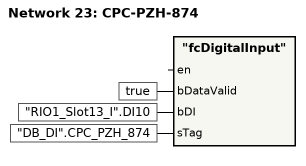
   "fcDigitalInput"(bDataValid := true, bDI := "RIO1_Slot13_I".DI10, sTag := "DB_DI".CPC_PZH_874);
END_REGION
END_FUNCTION_BLOCK

FUNCTION "fcDigitalInput" : Void
{ S7_Optimized_Access := 'TRUE' }
AUTHOR : Heaten
VERSION : 0.1
   VAR_INPUT 
      bDataValid : Bool;   // 1 = valid signal, 0 = invalid signal
      bDI : Bool;   // DI channel
   END_VAR

   VAR_IN_OUT 
      sTag : "stDigitalInput";
   END_VAR


BEGIN
	// Validate a digital input signal
	
	#sTag.bError := NOT(#bDataValid);
	
	IF #sTag.bError = TRUE THEN
	    #sTag.bValue := #sTag.bValueOnError;
	ELSE
	    #sTag.bValue := #bDI;
	END_IF;
END_FUNCTION

FUNCTION "fcAnalogInput" : Void
{ S7_Optimized_Access := 'TRUE' }
AUTHOR : Heaten
VERSION : 0.1
   VAR_INPUT 
      bValidData : Bool;
      iAI : Int;
      fOffset : Real;
   END_VAR

   VAR_OUTPUT 
      fEngValue : Real;
   END_VAR

   VAR_IN_OUT 
      sTag : "stAnalogInput";
   END_VAR

   VAR_TEMP 
      fSlope : Real;
      fIntercept : Real;
      fValue : Real;
   END_VAR


BEGIN
	// This is a version of fbAnalogInput that does not cache the scaling factors
	// An FB version takes 315 bytes per instance :(
	
	#sTag.Raw.iValue := #iAI;
	#sTag.Raw.bFault := NOT #bValidData;
	
	// Scaling
	IF NOT #bValidData THEN
	    #sTag.Eng.bError := TRUE;
	    #sTag.Eng.fValue := "NaN"();
	ELSE
	    #sTag.Eng.bError := FALSE;
	    IF #sTag.Raw.iMax <> 0 OR #sTag.Raw.iMin <> 0 THEN
	        #fSlope := (#sTag.Eng.fMax - #sTag.Eng.fMin) / INT_TO_REAL(#sTag.Raw.iMax - #sTag.Raw.iMin);
	    END_IF;
	    #fIntercept := #sTag.Eng.fMax - #fSlope*INT_TO_REAL(#sTag.Raw.iMax);
	    #fValue := INT_TO_REAL(#iAI)*#fSlope + #fIntercept + #fOffset;
	    // Apply limiting, if enabled
	    "fcCalcAssign"(fValue := #fValue, sTag := #sTag.Eng);
	END_IF;
	
	// Local output
	#fEngValue := #sTag.Eng.fValue;
	
END_FUNCTION

FUNCTION "fcCalcAssign" : Void

{ S7_Optimized_Access := 'TRUE' }
VERSION : 0.1
VAR_INPUT
  fValue : Real;
END_VAR

VAR_OUTPUT

END_VAR

VAR_IN_OUT
  sTag : "stCalcValue";
END_VAR

VAR_TEMP

END_VAR

VAR CONSTANT

END_VAR


BEGIN
	// When assigning to a calc value, set sTag.fValue and bits
	
	IF "isNaN"(#fValue) THEN
	    // Set error on NaN in
	    #sTag.bError := TRUE;
	    #sTag.fValue := #fValue;
	    #sTag.bLimited := FALSE;
	ELSE
	    // Valid values
	    #sTag.bError := FALSE;
	    IF #sTag.bCheckLimits = TRUE THEN
	        // With limitation
	        #sTag.fValue := LIMIT(IN := #fValue, MN := #sTag.fMin, MX := #sTag.fMax);
	        #sTag.bLimited := #fValue <> #sTag.fValue;
	    ELSE
	        // Without limitation
	        #sTag.fValue := #fValue;
	        #sTag.bLimited := FALSE;
	    END_IF;
	END_IF;
END_FUNCTION

FUNCTION "isNaN" : Bool   // FC19, FBD
TITLE = isNaN
{ S7_Optimized_Access := 'TRUE' }
VERSION : 0.1
// Returns TRUE if a REAL is NaN
// stored: AutoNumber true, IsIECCheckEnabled false, SetENOAutomatically false, UDAEnableTagReadback false
   VAR_INPUT
      In : Real;
   END_VAR
BEGIN

REGION Network 1
   // NOT_OK is a compiler builtin, but not available in SCL
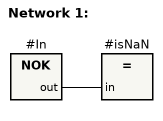
   // no SCL statement known for NOK: written as a call
   #isNaN := NOK(#In);
END_REGION
END_FUNCTION

FUNCTION_BLOCK "AnalogInputProcessing"   // FB37, FBD
TITLE = Handle analog inputs
{ S7_Optimized_Access := 'TRUE' }
AUTHOR : Heaten
VERSION : 0.1
// Map & scale analog inputs
// stored: AutoNumber true, IsIECCheckEnabled false, IsRetainMemResEnabled false, MemoryReserve 0, SetENOAutomatically false, UDAEnableTagReadback false
   VAR
      bHere : Bool;
   END_VAR
   VAR_TEMP
      fDummy : Real;
      fMaxWindingTemperature : Real;
      HBL_PT_05 : Real;
   END_VAR
   VAR_TEMP   // added for the SCL form of the ladder/FBD networks
      _w1 : Bool;
   END_VAR
BEGIN

REGION Network 1: HBL_TT_03 Oil sump oil temperature
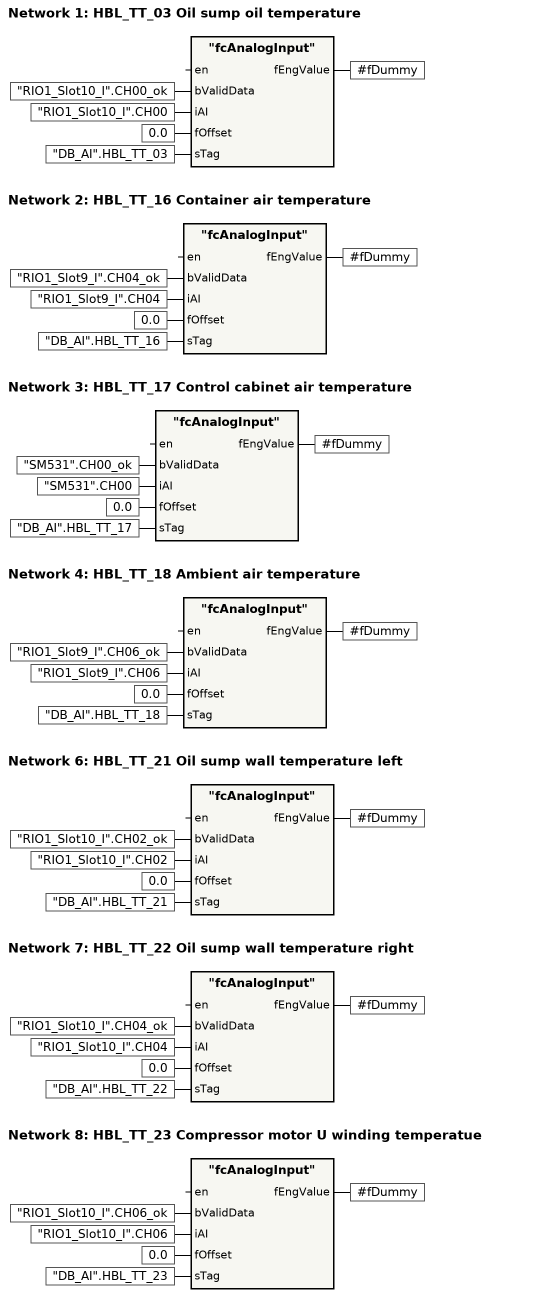
   "fcAnalogInput"(bValidData := "RIO1_Slot10_I".CH00_ok,
                   iAI := "RIO1_Slot10_I".CH00,
                   fOffset := 0.0,
                   sTag := "DB_AI".HBL_TT_03,
                   fEngValue => #fDummy);
END_REGION

REGION Network 2: HBL_TT_16 Container air temperature
   "fcAnalogInput"(bValidData := "RIO1_Slot9_I".CH04_ok,
                   iAI := "RIO1_Slot9_I".CH04,
                   fOffset := 0.0,
                   sTag := "DB_AI".HBL_TT_16,
                   fEngValue => #fDummy);
END_REGION

REGION Network 3: HBL_TT_17 Control cabinet air temperature
   "fcAnalogInput"(bValidData := "SM531".CH00_ok,
                   iAI := "SM531".CH00,
                   fOffset := 0.0,
                   sTag := "DB_AI".HBL_TT_17,
                   fEngValue => #fDummy);
END_REGION

REGION Network 4: HBL_TT_18 Ambient air temperature
   "fcAnalogInput"(bValidData := "RIO1_Slot9_I".CH06_ok,
                   iAI := "RIO1_Slot9_I".CH06,
                   fOffset := 0.0,
                   sTag := "DB_AI".HBL_TT_18,
                   fEngValue => #fDummy);
END_REGION

REGION Network 5: HBL_TT_19 Main inverter temperature
   // ##This is a fieldbus value. get from inverter, if we need it.
END_REGION

REGION Network 6: HBL_TT_21 Oil sump wall temperature left
   "fcAnalogInput"(bValidData := "RIO1_Slot10_I".CH02_ok,
                   iAI := "RIO1_Slot10_I".CH02,
                   fOffset := 0.0,
                   sTag := "DB_AI".HBL_TT_21,
                   fEngValue => #fDummy);
END_REGION

REGION Network 7: HBL_TT_22 Oil sump wall temperature right
   "fcAnalogInput"(bValidData := "RIO1_Slot10_I".CH04_ok,
                   iAI := "RIO1_Slot10_I".CH04,
                   fOffset := 0.0,
                   sTag := "DB_AI".HBL_TT_22,
                   fEngValue => #fDummy);
END_REGION

REGION Network 8: HBL_TT_23 Compressor motor U winding temperatue
   "fcAnalogInput"(bValidData := "RIO1_Slot10_I".CH06_ok,
                   iAI := "RIO1_Slot10_I".CH06,
                   fOffset := 0.0,
                   sTag := "DB_AI".HBL_TT_23,
                   fEngValue => #fDummy);
END_REGION

REGION Network 9: HBL_TT_24 Compressor motor V winding temperature
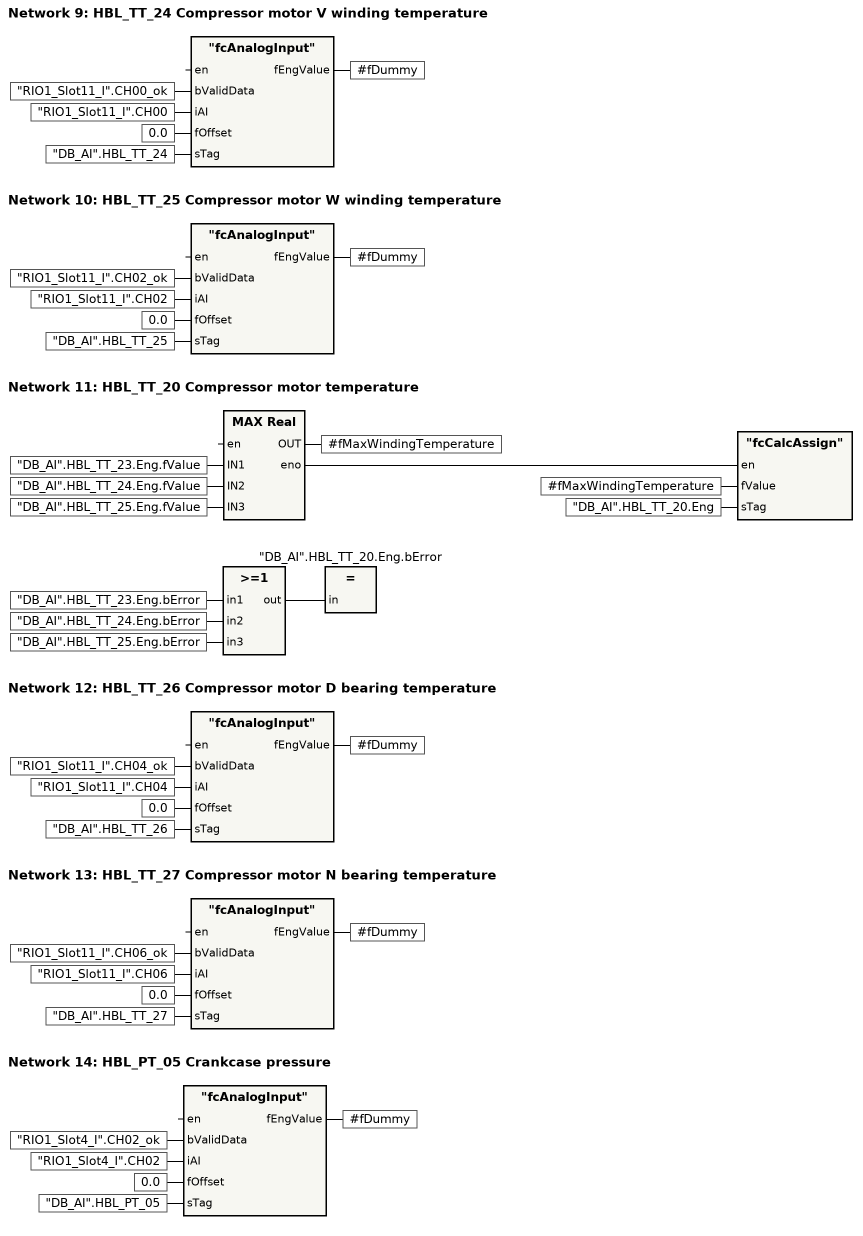
   "fcAnalogInput"(bValidData := "RIO1_Slot11_I".CH00_ok,
                   iAI := "RIO1_Slot11_I".CH00,
                   fOffset := 0.0,
                   sTag := "DB_AI".HBL_TT_24,
                   fEngValue => #fDummy);
END_REGION

REGION Network 10: HBL_TT_25 Compressor motor W winding temperature
   "fcAnalogInput"(bValidData := "RIO1_Slot11_I".CH02_ok,
                   iAI := "RIO1_Slot11_I".CH02,
                   fOffset := 0.0,
                   sTag := "DB_AI".HBL_TT_25,
                   fEngValue => #fDummy);
END_REGION

REGION Network 11: HBL_TT_20 Compressor motor temperature
   // MAX of any of the winding temperatures. If there is only one motor temperature, eg one PTC, use HBL-TT-20 as the analog input object
   // The individual winding temperatures are not used in the program (but are available for monitoring & logging)
   #fMaxWindingTemperature := MAX(IN1 := "DB_AI".HBL_TT_23.Eng.fValue, IN2 := "DB_AI".HBL_TT_24.Eng.fValue, IN3 := "DB_AI".HBL_TT_25.Eng.fValue);
   "fcCalcAssign"(fValue := #fMaxWindingTemperature, sTag := "DB_AI".HBL_TT_20.Eng);
   "DB_AI".HBL_TT_20.Eng.bError := "DB_AI".HBL_TT_23.Eng.bError OR "DB_AI".HBL_TT_24.Eng.bError OR "DB_AI".HBL_TT_25.Eng.bError;
END_REGION

REGION Network 12: HBL_TT_26 Compressor motor D bearing temperature
   "fcAnalogInput"(bValidData := "RIO1_Slot11_I".CH04_ok,
                   iAI := "RIO1_Slot11_I".CH04,
                   fOffset := 0.0,
                   sTag := "DB_AI".HBL_TT_26,
                   fEngValue => #fDummy);
END_REGION

REGION Network 13: HBL_TT_27 Compressor motor N bearing temperature
   "fcAnalogInput"(bValidData := "RIO1_Slot11_I".CH06_ok,
                   iAI := "RIO1_Slot11_I".CH06,
                   fOffset := 0.0,
                   sTag := "DB_AI".HBL_TT_27,
                   fEngValue => #fDummy);
END_REGION

REGION Network 14: HBL_PT_05 Crankcase pressure
   "fcAnalogInput"(bValidData := "RIO1_Slot4_I".CH02_ok,
                   iAI := "RIO1_Slot4_I".CH02,
                   fOffset := 0.0,
                   sTag := "DB_AI".HBL_PT_05,
                   fEngValue => #fDummy);
END_REGION

REGION Network 15: HBL_CT_01 Gas detector
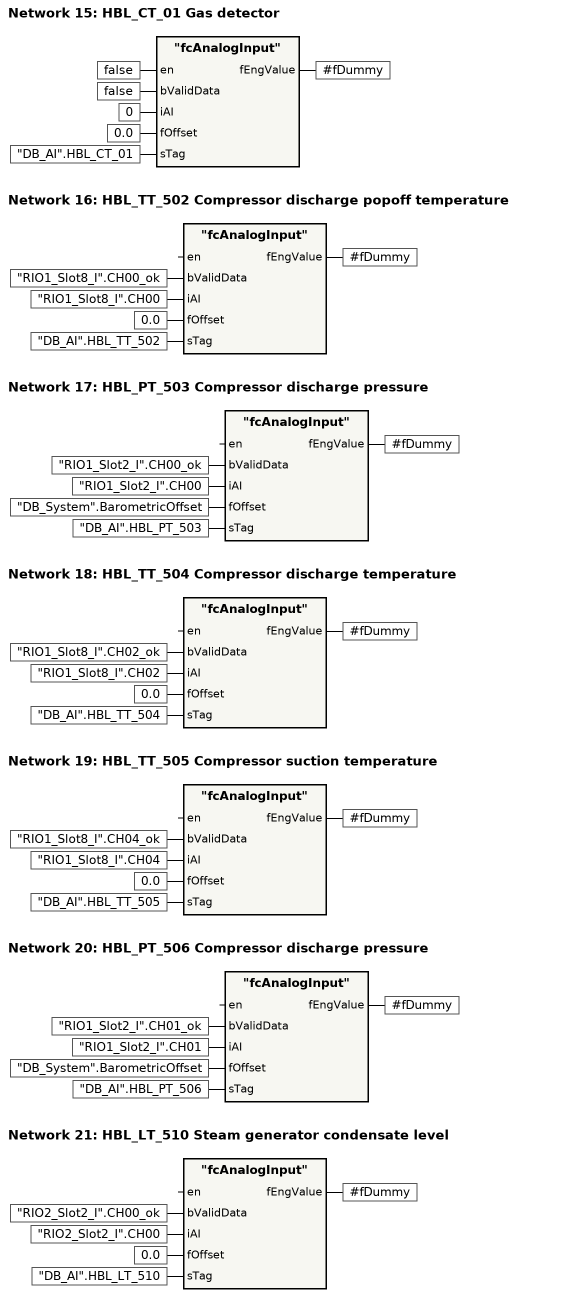
   IF false THEN
       "fcAnalogInput"(bValidData := false,
                       iAI := 0,
                       fOffset := 0.0,
                       sTag := "DB_AI".HBL_CT_01,
                       fEngValue => #fDummy);
   END_IF;
END_REGION

REGION Network 16: HBL_TT_502 Compressor discharge popoff temperature
   "fcAnalogInput"(bValidData := "RIO1_Slot8_I".CH00_ok,
                   iAI := "RIO1_Slot8_I".CH00,
                   fOffset := 0.0,
                   sTag := "DB_AI".HBL_TT_502,
                   fEngValue => #fDummy);
END_REGION

REGION Network 17: HBL_PT_503 Compressor discharge pressure
   "fcAnalogInput"(bValidData := "RIO1_Slot2_I".CH00_ok,
                   iAI := "RIO1_Slot2_I".CH00,
                   fOffset := "DB_System".BarometricOffset,
                   sTag := "DB_AI".HBL_PT_503,
                   fEngValue => #fDummy);
END_REGION

REGION Network 18: HBL_TT_504 Compressor discharge temperature
   "fcAnalogInput"(bValidData := "RIO1_Slot8_I".CH02_ok,
                   iAI := "RIO1_Slot8_I".CH02,
                   fOffset := 0.0,
                   sTag := "DB_AI".HBL_TT_504,
                   fEngValue => #fDummy);
END_REGION

REGION Network 19: HBL_TT_505 Compressor suction temperature
   "fcAnalogInput"(bValidData := "RIO1_Slot8_I".CH04_ok,
                   iAI := "RIO1_Slot8_I".CH04,
                   fOffset := 0.0,
                   sTag := "DB_AI".HBL_TT_505,
                   fEngValue => #fDummy);
END_REGION

REGION Network 20: HBL_PT_506 Compressor discharge pressure
   "fcAnalogInput"(bValidData := "RIO1_Slot2_I".CH01_ok,
                   iAI := "RIO1_Slot2_I".CH01,
                   fOffset := "DB_System".BarometricOffset,
                   sTag := "DB_AI".HBL_PT_506,
                   fEngValue => #fDummy);
END_REGION

REGION Network 21: HBL_LT_510 Steam generator condensate level
   "fcAnalogInput"(bValidData := "RIO2_Slot2_I".CH00_ok,
                   iAI := "RIO2_Slot2_I".CH00,
                   fOffset := 0.0,
                   sTag := "DB_AI".HBL_LT_510,
                   fEngValue => #fDummy);
END_REGION

REGION Network 22: HBL_PT_511 Heat sink discharge pressure
   // Local or remote
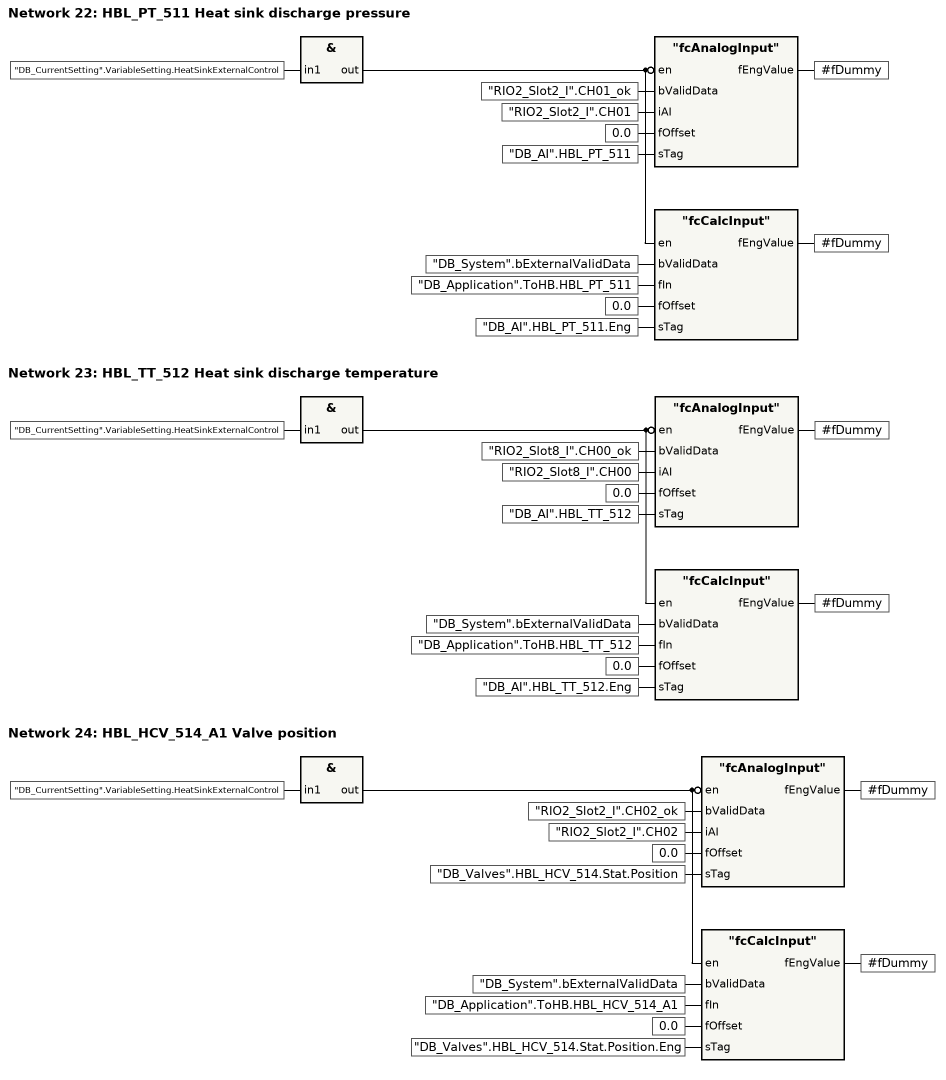
   #_w1 := "DB_CurrentSetting".VariableSetting.HeatSinkExternalControl;
   IF NOT "DB_CurrentSetting".VariableSetting.HeatSinkExternalControl THEN
       "fcAnalogInput"(bValidData := "RIO2_Slot2_I".CH01_ok,
                       iAI := "RIO2_Slot2_I".CH01,
                       fOffset := 0.0,
                       sTag := "DB_AI".HBL_PT_511,
                       fEngValue => #fDummy);
   END_IF;
   IF #_w1 THEN
       "fcCalcInput"(bValidData := "DB_System".bExternalValidData,
                     fIn := "DB_Application".ToHB.HBL_PT_511,
                     fOffset := 0.0,
                     sTag := "DB_AI".HBL_PT_511.Eng,
                     fEngValue => #fDummy);
   END_IF;
END_REGION

REGION Network 23: HBL_TT_512 Heat sink discharge temperature
   // Local or remote
   #_w1 := "DB_CurrentSetting".VariableSetting.HeatSinkExternalControl;
   IF NOT "DB_CurrentSetting".VariableSetting.HeatSinkExternalControl THEN
       "fcAnalogInput"(bValidData := "RIO2_Slot8_I".CH00_ok,
                       iAI := "RIO2_Slot8_I".CH00,
                       fOffset := 0.0,
                       sTag := "DB_AI".HBL_TT_512,
                       fEngValue => #fDummy);
   END_IF;
   IF #_w1 THEN
       "fcCalcInput"(bValidData := "DB_System".bExternalValidData,
                     fIn := "DB_Application".ToHB.HBL_TT_512,
                     fOffset := 0.0,
                     sTag := "DB_AI".HBL_TT_512.Eng,
                     fEngValue => #fDummy);
   END_IF;
END_REGION

REGION Network 24: HBL_HCV_514_A1 Valve position
   // Local or remote
   #_w1 := "DB_CurrentSetting".VariableSetting.HeatSinkExternalControl;
   IF NOT "DB_CurrentSetting".VariableSetting.HeatSinkExternalControl THEN
       "fcAnalogInput"(bValidData := "RIO2_Slot2_I".CH02_ok,
                       iAI := "RIO2_Slot2_I".CH02,
                       fOffset := 0.0,
                       sTag := "DB_Valves".HBL_HCV_514.Stat.Position,
                       fEngValue => #fDummy);
   END_IF;
   IF #_w1 THEN
       "fcCalcInput"(bValidData := "DB_System".bExternalValidData,
                     fIn := "DB_Application".ToHB.HBL_HCV_514_A1,
                     fOffset := 0.0,
                     sTag := "DB_Valves".HBL_HCV_514.Stat.Position.Eng,
                     fEngValue => #fDummy);
   END_IF;
END_REGION

REGION Network 25: HBL_HCV_515_A1 Heat sink condensate blowdown valve position
   // Local or remote
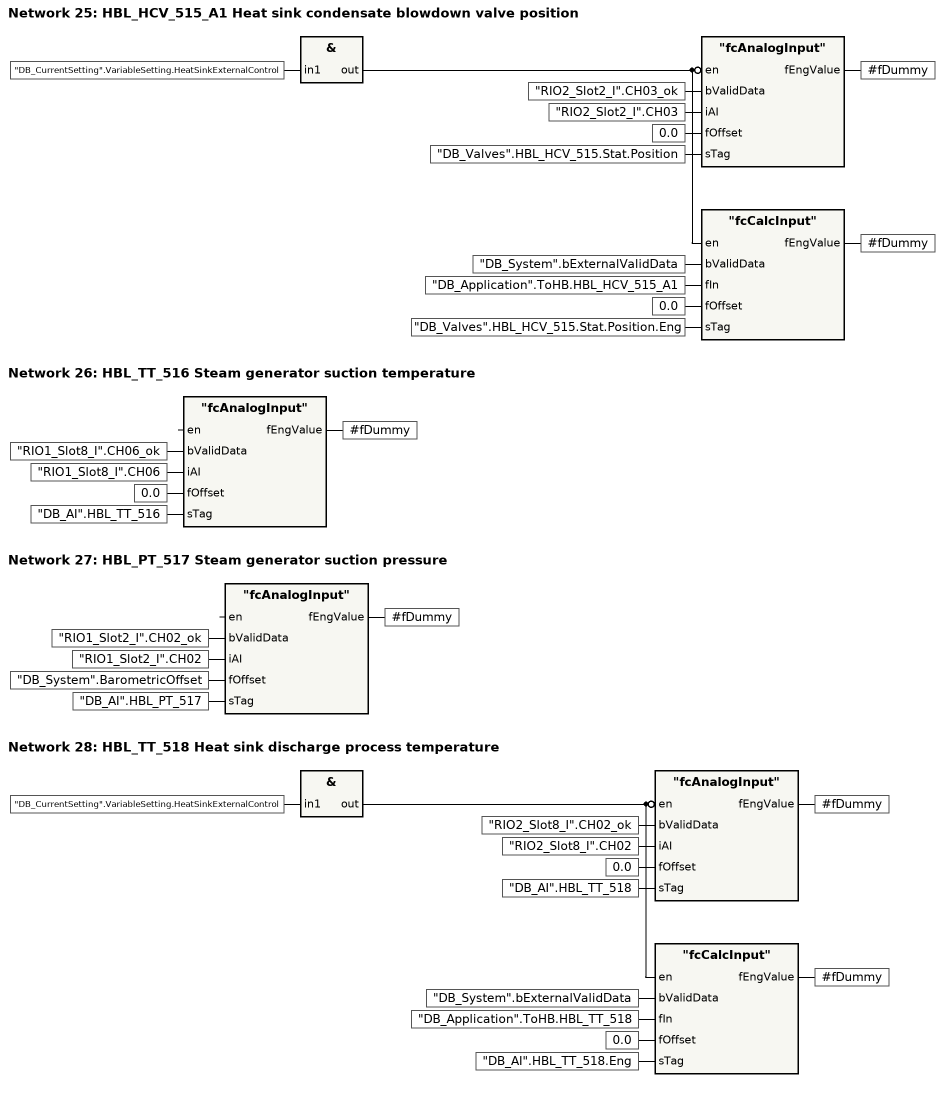
   #_w1 := "DB_CurrentSetting".VariableSetting.HeatSinkExternalControl;
   IF NOT "DB_CurrentSetting".VariableSetting.HeatSinkExternalControl THEN
       "fcAnalogInput"(bValidData := "RIO2_Slot2_I".CH03_ok,
                       iAI := "RIO2_Slot2_I".CH03,
                       fOffset := 0.0,
                       sTag := "DB_Valves".HBL_HCV_515.Stat.Position,
                       fEngValue => #fDummy);
   END_IF;
   IF #_w1 THEN
       "fcCalcInput"(bValidData := "DB_System".bExternalValidData,
                     fIn := "DB_Application".ToHB.HBL_HCV_515_A1,
                     fOffset := 0.0,
                     sTag := "DB_Valves".HBL_HCV_515.Stat.Position.Eng,
                     fEngValue => #fDummy);
   END_IF;
END_REGION

REGION Network 26: HBL_TT_516 Steam generator suction temperature
   "fcAnalogInput"(bValidData := "RIO1_Slot8_I".CH06_ok,
                   iAI := "RIO1_Slot8_I".CH06,
                   fOffset := 0.0,
                   sTag := "DB_AI".HBL_TT_516,
                   fEngValue => #fDummy);
END_REGION

REGION Network 27: HBL_PT_517 Steam generator suction pressure
   "fcAnalogInput"(bValidData := "RIO1_Slot2_I".CH02_ok,
                   iAI := "RIO1_Slot2_I".CH02,
                   fOffset := "DB_System".BarometricOffset,
                   sTag := "DB_AI".HBL_PT_517,
                   fEngValue => #fDummy);
END_REGION

REGION Network 28: HBL_TT_518 Heat sink discharge process temperature
   // Local or remote
   #_w1 := "DB_CurrentSetting".VariableSetting.HeatSinkExternalControl;
   IF NOT "DB_CurrentSetting".VariableSetting.HeatSinkExternalControl THEN
       "fcAnalogInput"(bValidData := "RIO2_Slot8_I".CH02_ok,
                       iAI := "RIO2_Slot8_I".CH02,
                       fOffset := 0.0,
                       sTag := "DB_AI".HBL_TT_518,
                       fEngValue => #fDummy);
   END_IF;
   IF #_w1 THEN
       "fcCalcInput"(bValidData := "DB_System".bExternalValidData,
                     fIn := "DB_Application".ToHB.HBL_TT_518,
                     fOffset := 0.0,
                     sTag := "DB_AI".HBL_TT_518.Eng,
                     fEngValue => #fDummy);
   END_IF;
END_REGION

REGION Network 29: HBL_PT_519 Heat sink discharge process pressure
   // Local or remote
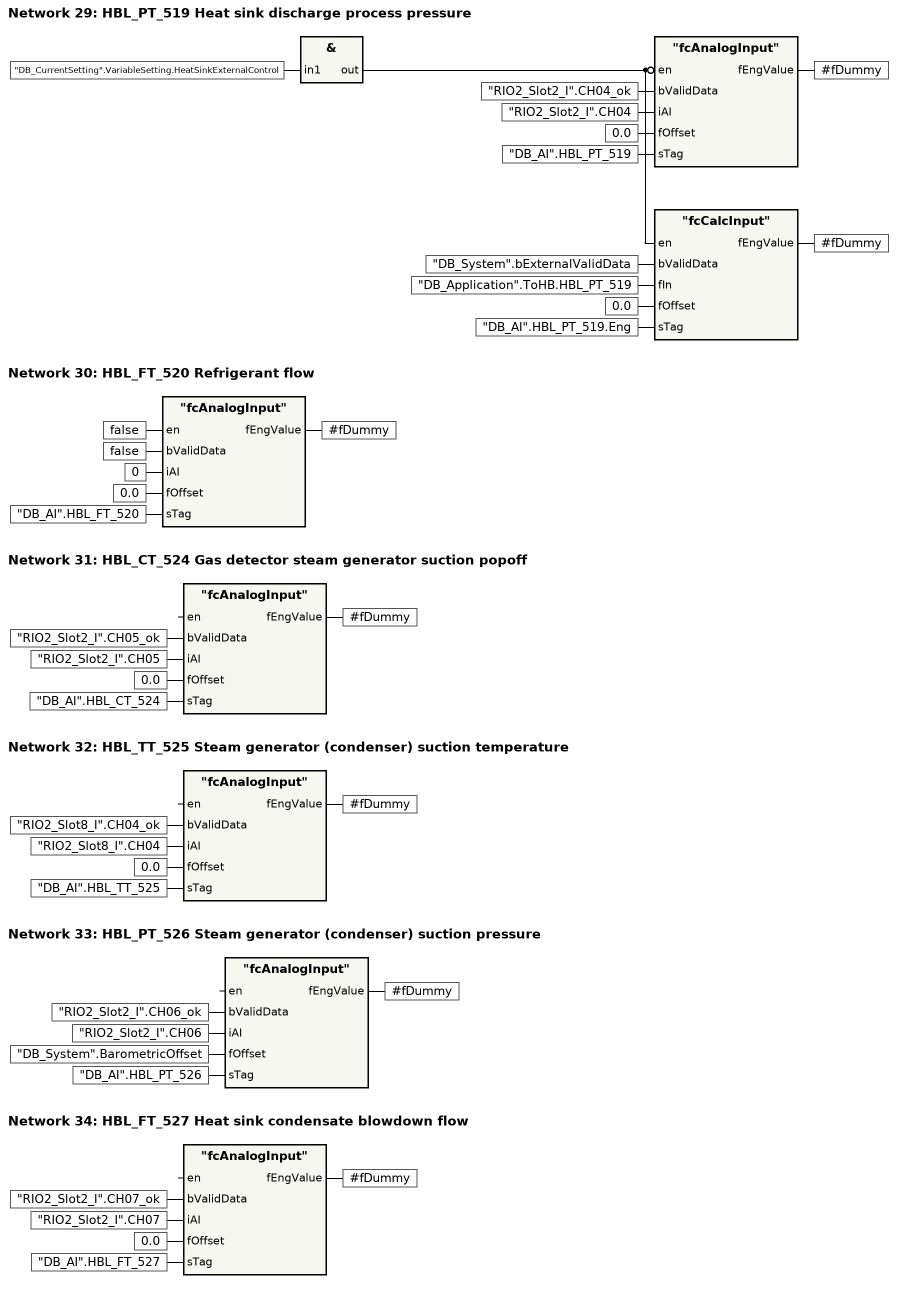
   #_w1 := "DB_CurrentSetting".VariableSetting.HeatSinkExternalControl;
   IF NOT "DB_CurrentSetting".VariableSetting.HeatSinkExternalControl THEN
       "fcAnalogInput"(bValidData := "RIO2_Slot2_I".CH04_ok,
                       iAI := "RIO2_Slot2_I".CH04,
                       fOffset := 0.0,
                       sTag := "DB_AI".HBL_PT_519,
                       fEngValue => #fDummy);
   END_IF;
   IF #_w1 THEN
       "fcCalcInput"(bValidData := "DB_System".bExternalValidData,
                     fIn := "DB_Application".ToHB.HBL_PT_519,
                     fOffset := 0.0,
                     sTag := "DB_AI".HBL_PT_519.Eng,
                     fEngValue => #fDummy);
   END_IF;
END_REGION

REGION Network 30: HBL_FT_520 Refrigerant flow
   // Not used in Offenau
   IF false THEN
       "fcAnalogInput"(bValidData := false,
                       iAI := 0,
                       fOffset := 0.0,
                       sTag := "DB_AI".HBL_FT_520,
                       fEngValue => #fDummy);
   END_IF;
END_REGION

REGION Network 31: HBL_CT_524 Gas detector steam generator suction popoff
   "fcAnalogInput"(bValidData := "RIO2_Slot2_I".CH05_ok,
                   iAI := "RIO2_Slot2_I".CH05,
                   fOffset := 0.0,
                   sTag := "DB_AI".HBL_CT_524,
                   fEngValue => #fDummy);
END_REGION

REGION Network 32: HBL_TT_525 Steam generator (condenser) suction temperature
   "fcAnalogInput"(bValidData := "RIO2_Slot8_I".CH04_ok,
                   iAI := "RIO2_Slot8_I".CH04,
                   fOffset := 0.0,
                   sTag := "DB_AI".HBL_TT_525,
                   fEngValue => #fDummy);
END_REGION

REGION Network 33: HBL_PT_526 Steam generator (condenser) suction pressure
   "fcAnalogInput"(bValidData := "RIO2_Slot2_I".CH06_ok,
                   iAI := "RIO2_Slot2_I".CH06,
                   fOffset := "DB_System".BarometricOffset,
                   sTag := "DB_AI".HBL_PT_526,
                   fEngValue => #fDummy);
END_REGION

REGION Network 34: HBL_FT_527 Heat sink condensate blowdown flow
   "fcAnalogInput"(bValidData := "RIO2_Slot2_I".CH07_ok,
                   iAI := "RIO2_Slot2_I".CH07,
                   fOffset := 0.0,
                   sTag := "DB_AI".HBL_FT_527,
                   fEngValue => #fDummy);
END_REGION

REGION Network 35: HBL_TT_530 Expansion valve B discharge temperature
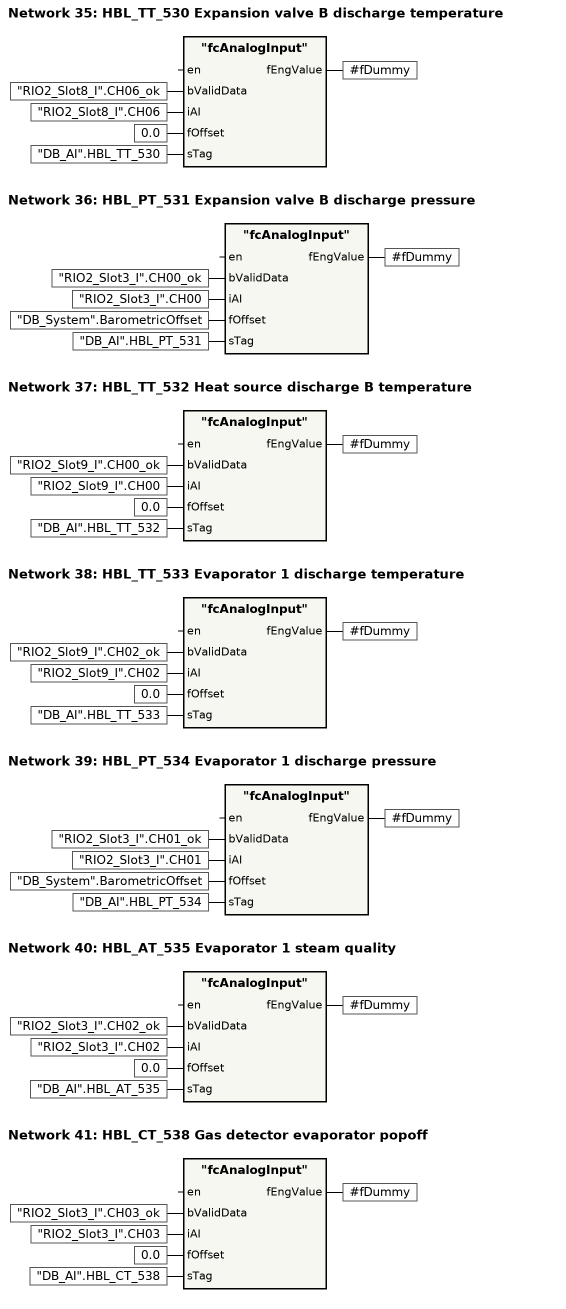
   "fcAnalogInput"(bValidData := "RIO2_Slot8_I".CH06_ok,
                   iAI := "RIO2_Slot8_I".CH06,
                   fOffset := 0.0,
                   sTag := "DB_AI".HBL_TT_530,
                   fEngValue => #fDummy);
END_REGION

REGION Network 36: HBL_PT_531 Expansion valve B discharge pressure
   // Convert from rel to abs
   "fcAnalogInput"(bValidData := "RIO2_Slot3_I".CH00_ok,
                   iAI := "RIO2_Slot3_I".CH00,
                   fOffset := "DB_System".BarometricOffset,
                   sTag := "DB_AI".HBL_PT_531,
                   fEngValue => #fDummy);
END_REGION

REGION Network 37: HBL_TT_532 Heat source discharge B temperature
   "fcAnalogInput"(bValidData := "RIO2_Slot9_I".CH00_ok,
                   iAI := "RIO2_Slot9_I".CH00,
                   fOffset := 0.0,
                   sTag := "DB_AI".HBL_TT_532,
                   fEngValue => #fDummy);
END_REGION

REGION Network 38: HBL_TT_533 Evaporator 1 discharge temperature
   "fcAnalogInput"(bValidData := "RIO2_Slot9_I".CH02_ok,
                   iAI := "RIO2_Slot9_I".CH02,
                   fOffset := 0.0,
                   sTag := "DB_AI".HBL_TT_533,
                   fEngValue => #fDummy);
END_REGION

REGION Network 39: HBL_PT_534 Evaporator 1 discharge pressure
   // Convert from rel to abs
   "fcAnalogInput"(bValidData := "RIO2_Slot3_I".CH01_ok,
                   iAI := "RIO2_Slot3_I".CH01,
                   fOffset := "DB_System".BarometricOffset,
                   sTag := "DB_AI".HBL_PT_534,
                   fEngValue => #fDummy);
END_REGION

REGION Network 40: HBL_AT_535 Evaporator 1 steam quality
   "fcAnalogInput"(bValidData := "RIO2_Slot3_I".CH02_ok,
                   iAI := "RIO2_Slot3_I".CH02,
                   fOffset := 0.0,
                   sTag := "DB_AI".HBL_AT_535,
                   fEngValue => #fDummy);
END_REGION

REGION Network 41: HBL_CT_538 Gas detector evaporator popoff
   "fcAnalogInput"(bValidData := "RIO2_Slot3_I".CH03_ok,
                   iAI := "RIO2_Slot3_I".CH03,
                   fOffset := 0.0,
                   sTag := "DB_AI".HBL_CT_538,
                   fEngValue => #fDummy);
END_REGION

REGION Network 42: HBL_TT_540 Expansion valve A discharge temperature
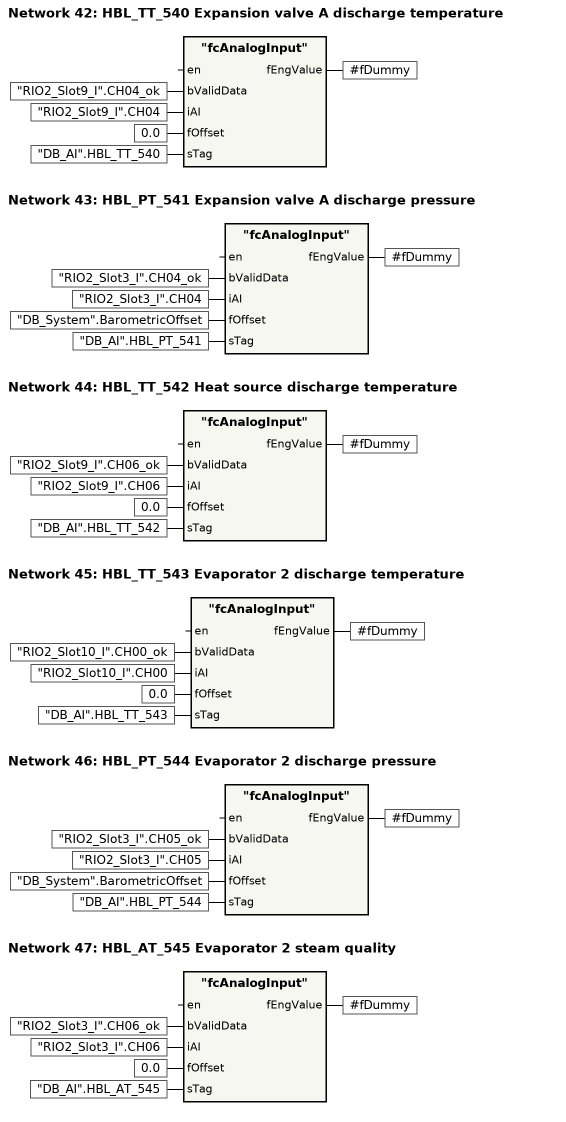
   "fcAnalogInput"(bValidData := "RIO2_Slot9_I".CH04_ok,
                   iAI := "RIO2_Slot9_I".CH04,
                   fOffset := 0.0,
                   sTag := "DB_AI".HBL_TT_540,
                   fEngValue => #fDummy);
END_REGION

REGION Network 43: HBL_PT_541 Expansion valve A discharge pressure
   "fcAnalogInput"(bValidData := "RIO2_Slot3_I".CH04_ok,
                   iAI := "RIO2_Slot3_I".CH04,
                   fOffset := "DB_System".BarometricOffset,
                   sTag := "DB_AI".HBL_PT_541,
                   fEngValue => #fDummy);
END_REGION

REGION Network 44: HBL_TT_542 Heat source discharge temperature
   "fcAnalogInput"(bValidData := "RIO2_Slot9_I".CH06_ok,
                   iAI := "RIO2_Slot9_I".CH06,
                   fOffset := 0.0,
                   sTag := "DB_AI".HBL_TT_542,
                   fEngValue => #fDummy);
END_REGION

REGION Network 45: HBL_TT_543 Evaporator 2 discharge temperature
   "fcAnalogInput"(bValidData := "RIO2_Slot10_I".CH00_ok,
                   iAI := "RIO2_Slot10_I".CH00,
                   fOffset := 0.0,
                   sTag := "DB_AI".HBL_TT_543,
                   fEngValue => #fDummy);
END_REGION

REGION Network 46: HBL_PT_544 Evaporator 2 discharge pressure
   "fcAnalogInput"(bValidData := "RIO2_Slot3_I".CH05_ok,
                   iAI := "RIO2_Slot3_I".CH05,
                   fOffset := "DB_System".BarometricOffset,
                   sTag := "DB_AI".HBL_PT_544,
                   fEngValue => #fDummy);
END_REGION

REGION Network 47: HBL_AT_545 Evaporator 2 steam quality
   "fcAnalogInput"(bValidData := "RIO2_Slot3_I".CH06_ok,
                   iAI := "RIO2_Slot3_I".CH06,
                   fOffset := 0.0,
                   sTag := "DB_AI".HBL_AT_545,
                   fEngValue => #fDummy);
END_REGION

REGION Network 48: HBL_TT_546 Heat source suction temperature
   // Local or remote
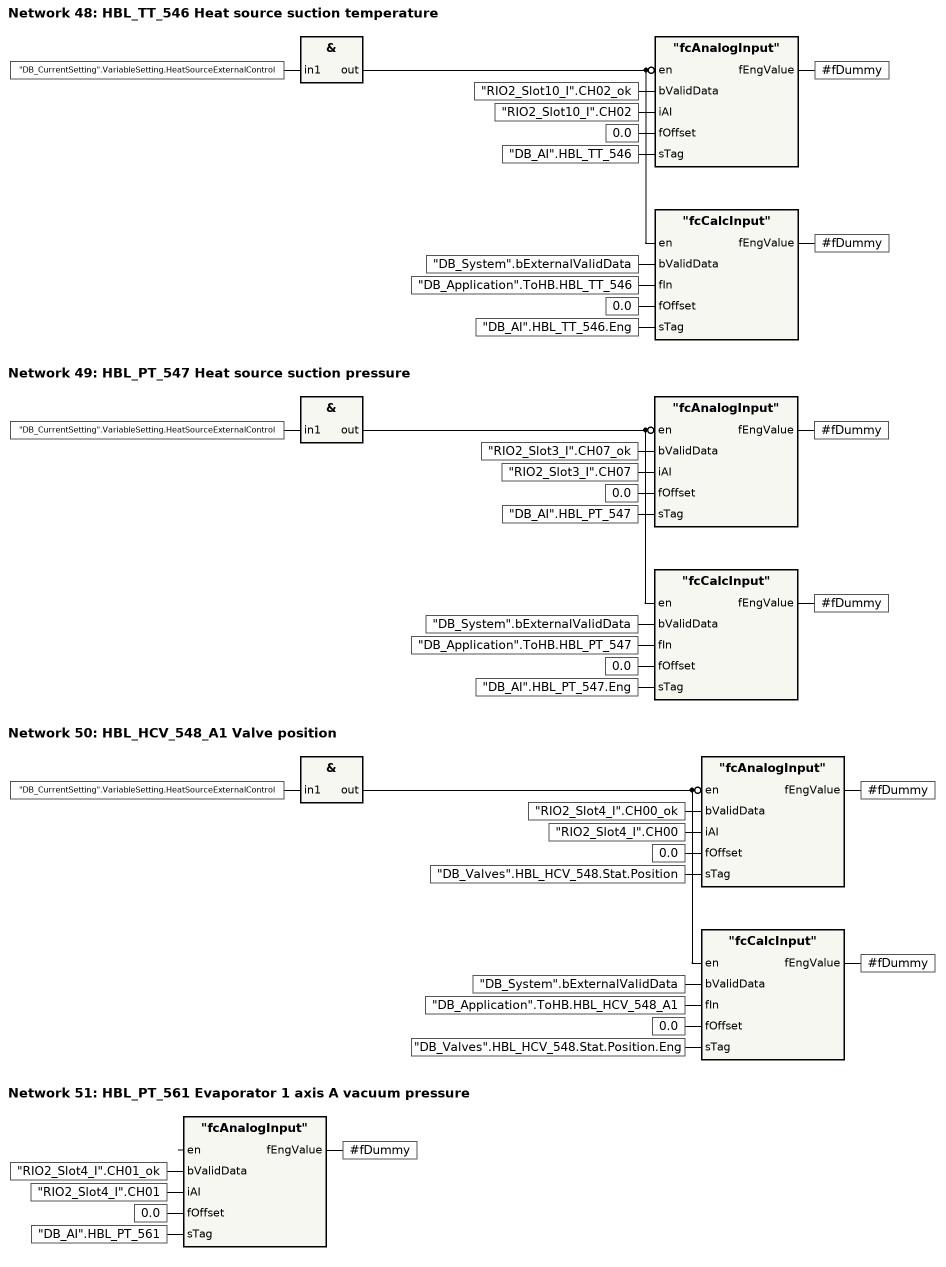
   #_w1 := "DB_CurrentSetting".VariableSetting.HeatSourceExternalControl;
   IF NOT "DB_CurrentSetting".VariableSetting.HeatSourceExternalControl THEN
       "fcAnalogInput"(bValidData := "RIO2_Slot10_I".CH02_ok,
                       iAI := "RIO2_Slot10_I".CH02,
                       fOffset := 0.0,
                       sTag := "DB_AI".HBL_TT_546,
                       fEngValue => #fDummy);
   END_IF;
   IF #_w1 THEN
       "fcCalcInput"(bValidData := "DB_System".bExternalValidData,
                     fIn := "DB_Application".ToHB.HBL_TT_546,
                     fOffset := 0.0,
                     sTag := "DB_AI".HBL_TT_546.Eng,
                     fEngValue => #fDummy);
   END_IF;
END_REGION

REGION Network 49: HBL_PT_547 Heat source suction pressure
   // Local or remote
   #_w1 := "DB_CurrentSetting".VariableSetting.HeatSourceExternalControl;
   IF NOT "DB_CurrentSetting".VariableSetting.HeatSourceExternalControl THEN
       "fcAnalogInput"(bValidData := "RIO2_Slot3_I".CH07_ok,
                       iAI := "RIO2_Slot3_I".CH07,
                       fOffset := 0.0,
                       sTag := "DB_AI".HBL_PT_547,
                       fEngValue => #fDummy);
   END_IF;
   IF #_w1 THEN
       "fcCalcInput"(bValidData := "DB_System".bExternalValidData,
                     fIn := "DB_Application".ToHB.HBL_PT_547,
                     fOffset := 0.0,
                     sTag := "DB_AI".HBL_PT_547.Eng,
                     fEngValue => #fDummy);
   END_IF;
END_REGION

REGION Network 50: HBL_HCV_548_A1 Valve position
   // Local or remote
   #_w1 := "DB_CurrentSetting".VariableSetting.HeatSourceExternalControl;
   IF NOT "DB_CurrentSetting".VariableSetting.HeatSourceExternalControl THEN
       "fcAnalogInput"(bValidData := "RIO2_Slot4_I".CH00_ok,
                       iAI := "RIO2_Slot4_I".CH00,
                       fOffset := 0.0,
                       sTag := "DB_Valves".HBL_HCV_548.Stat.Position,
                       fEngValue => #fDummy);
   END_IF;
   IF #_w1 THEN
       "fcCalcInput"(bValidData := "DB_System".bExternalValidData,
                     fIn := "DB_Application".ToHB.HBL_HCV_548_A1,
                     fOffset := 0.0,
                     sTag := "DB_Valves".HBL_HCV_548.Stat.Position.Eng,
                     fEngValue => #fDummy);
   END_IF;
END_REGION

REGION Network 51: HBL_PT_561 Evaporator 1 axis A vacuum pressure
   "fcAnalogInput"(bValidData := "RIO2_Slot4_I".CH01_ok,
                   iAI := "RIO2_Slot4_I".CH01,
                   fOffset := 0.0,
                   sTag := "DB_AI".HBL_PT_561,
                   fEngValue => #fDummy);
END_REGION

REGION Network 52: HBL_PT_562 Evaporator 2 axis A vacuum pressure
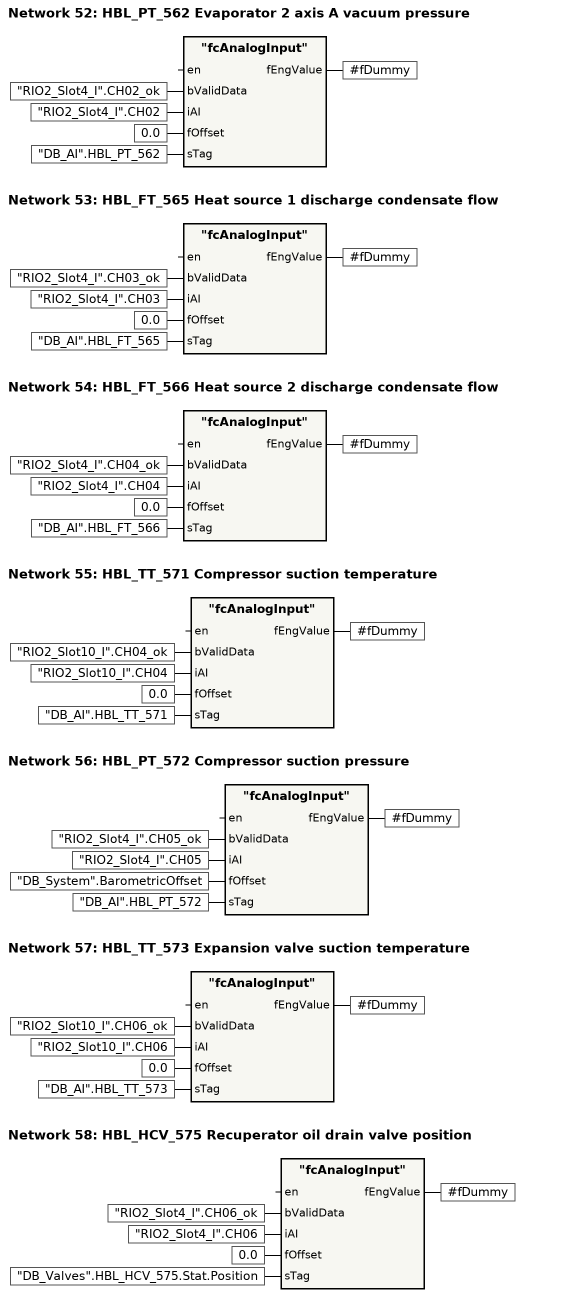
   "fcAnalogInput"(bValidData := "RIO2_Slot4_I".CH02_ok,
                   iAI := "RIO2_Slot4_I".CH02,
                   fOffset := 0.0,
                   sTag := "DB_AI".HBL_PT_562,
                   fEngValue => #fDummy);
END_REGION

REGION Network 53: HBL_FT_565 Heat source 1 discharge condensate flow
   "fcAnalogInput"(bValidData := "RIO2_Slot4_I".CH03_ok,
                   iAI := "RIO2_Slot4_I".CH03,
                   fOffset := 0.0,
                   sTag := "DB_AI".HBL_FT_565,
                   fEngValue => #fDummy);
END_REGION

REGION Network 54: HBL_FT_566 Heat source 2 discharge condensate flow
   "fcAnalogInput"(bValidData := "RIO2_Slot4_I".CH04_ok,
                   iAI := "RIO2_Slot4_I".CH04,
                   fOffset := 0.0,
                   sTag := "DB_AI".HBL_FT_566,
                   fEngValue => #fDummy);
END_REGION

REGION Network 55: HBL_TT_571 Compressor suction temperature
   "fcAnalogInput"(bValidData := "RIO2_Slot10_I".CH04_ok,
                   iAI := "RIO2_Slot10_I".CH04,
                   fOffset := 0.0,
                   sTag := "DB_AI".HBL_TT_571,
                   fEngValue => #fDummy);
END_REGION

REGION Network 56: HBL_PT_572 Compressor suction pressure
   "fcAnalogInput"(bValidData := "RIO2_Slot4_I".CH05_ok,
                   iAI := "RIO2_Slot4_I".CH05,
                   fOffset := "DB_System".BarometricOffset,
                   sTag := "DB_AI".HBL_PT_572,
                   fEngValue => #fDummy);
END_REGION

REGION Network 57: HBL_TT_573 Expansion valve suction temperature
   "fcAnalogInput"(bValidData := "RIO2_Slot10_I".CH06_ok,
                   iAI := "RIO2_Slot10_I".CH06,
                   fOffset := 0.0,
                   sTag := "DB_AI".HBL_TT_573,
                   fEngValue => #fDummy);
END_REGION

REGION Network 58: HBL_HCV_575 Recuperator oil drain valve position
   "fcAnalogInput"(bValidData := "RIO2_Slot4_I".CH06_ok,
                   iAI := "RIO2_Slot4_I".CH06,
                   fOffset := 0.0,
                   sTag := "DB_Valves".HBL_HCV_575.Stat.Position,
                   fEngValue => #fDummy);
END_REGION

REGION Network 59: HBL_HCV_576 Expansion Valve A position
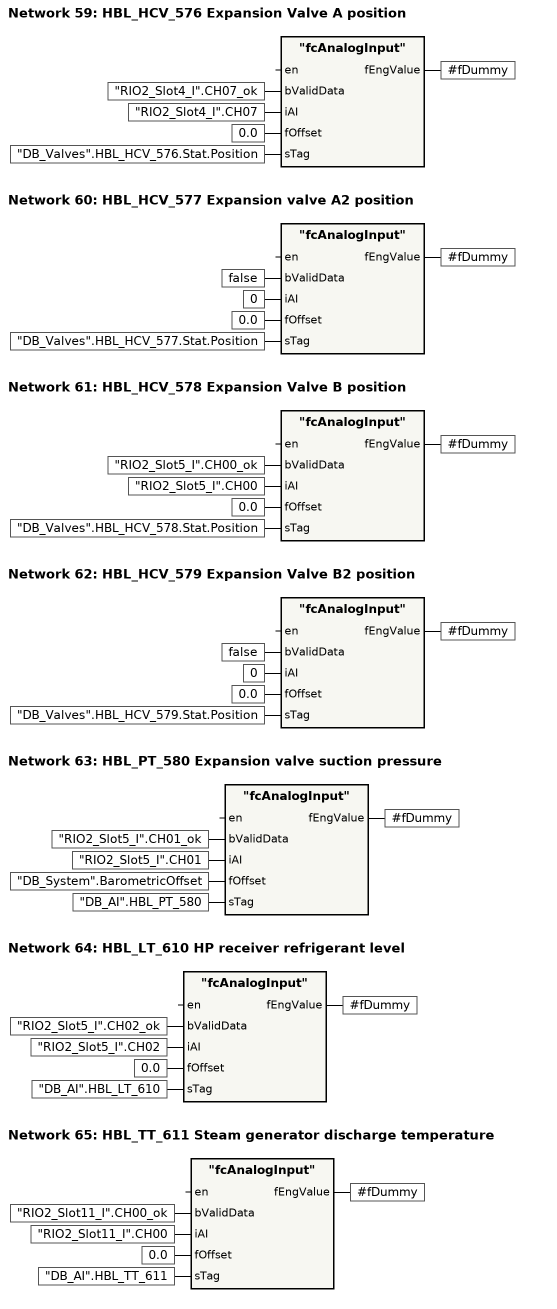
   "fcAnalogInput"(bValidData := "RIO2_Slot4_I".CH07_ok,
                   iAI := "RIO2_Slot4_I".CH07,
                   fOffset := 0.0,
                   sTag := "DB_Valves".HBL_HCV_576.Stat.Position,
                   fEngValue => #fDummy);
END_REGION

REGION Network 60: HBL_HCV_577 Expansion valve A2 position
   "fcAnalogInput"(bValidData := false,
                   iAI := 0,
                   fOffset := 0.0,
                   sTag := "DB_Valves".HBL_HCV_577.Stat.Position,
                   fEngValue => #fDummy);
END_REGION

REGION Network 61: HBL_HCV_578 Expansion Valve B position
   "fcAnalogInput"(bValidData := "RIO2_Slot5_I".CH00_ok,
                   iAI := "RIO2_Slot5_I".CH00,
                   fOffset := 0.0,
                   sTag := "DB_Valves".HBL_HCV_578.Stat.Position,
                   fEngValue => #fDummy);
END_REGION

REGION Network 62: HBL_HCV_579 Expansion Valve B2 position
   "fcAnalogInput"(bValidData := false,
                   iAI := 0,
                   fOffset := 0.0,
                   sTag := "DB_Valves".HBL_HCV_579.Stat.Position,
                   fEngValue => #fDummy);
END_REGION

REGION Network 63: HBL_PT_580 Expansion valve suction pressure
   "fcAnalogInput"(bValidData := "RIO2_Slot5_I".CH01_ok,
                   iAI := "RIO2_Slot5_I".CH01,
                   fOffset := "DB_System".BarometricOffset,
                   sTag := "DB_AI".HBL_PT_580,
                   fEngValue => #fDummy);
END_REGION

REGION Network 64: HBL_LT_610 HP receiver refrigerant level
   "fcAnalogInput"(bValidData := "RIO2_Slot5_I".CH02_ok,
                   iAI := "RIO2_Slot5_I".CH02,
                   fOffset := 0.0,
                   sTag := "DB_AI".HBL_LT_610,
                   fEngValue => #fDummy);
END_REGION

REGION Network 65: HBL_TT_611 Steam generator discharge temperature
   "fcAnalogInput"(bValidData := "RIO2_Slot11_I".CH00_ok,
                   iAI := "RIO2_Slot11_I".CH00,
                   fOffset := 0.0,
                   sTag := "DB_AI".HBL_TT_611,
                   fEngValue => #fDummy);
END_REGION

REGION Network 66: HBL_PT_612 Steam generator discharge pressure
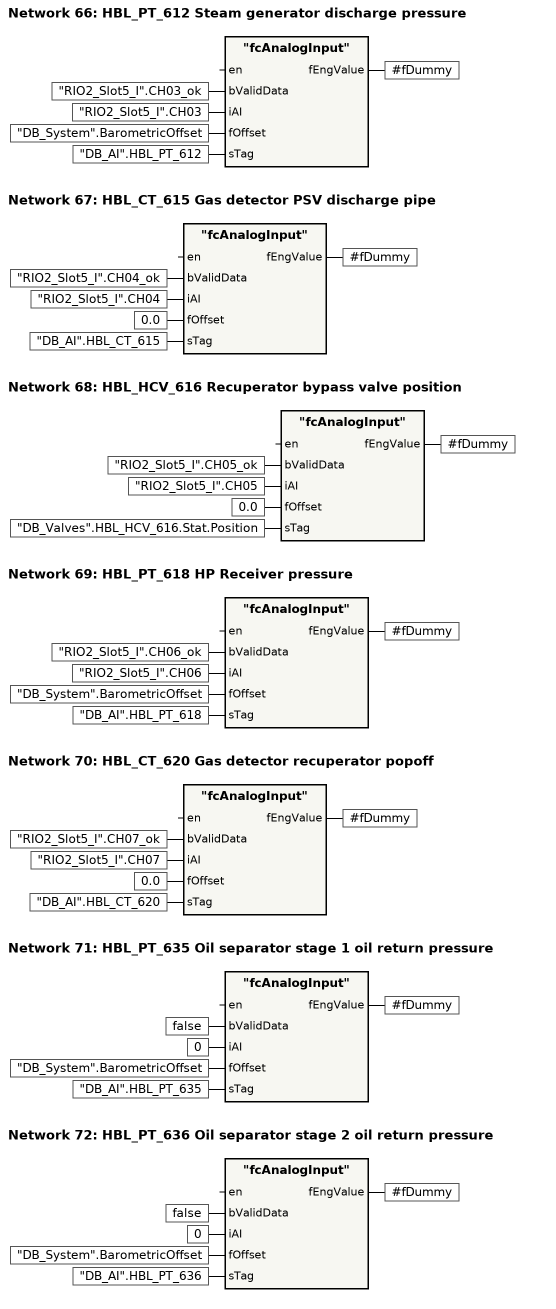
   "fcAnalogInput"(bValidData := "RIO2_Slot5_I".CH03_ok,
                   iAI := "RIO2_Slot5_I".CH03,
                   fOffset := "DB_System".BarometricOffset,
                   sTag := "DB_AI".HBL_PT_612,
                   fEngValue => #fDummy);
END_REGION

REGION Network 67: HBL_CT_615 Gas detector PSV discharge pipe
   "fcAnalogInput"(bValidData := "RIO2_Slot5_I".CH04_ok,
                   iAI := "RIO2_Slot5_I".CH04,
                   fOffset := 0.0,
                   sTag := "DB_AI".HBL_CT_615,
                   fEngValue => #fDummy);
END_REGION

REGION Network 68: HBL_HCV_616 Recuperator bypass valve position
   "fcAnalogInput"(bValidData := "RIO2_Slot5_I".CH05_ok,
                   iAI := "RIO2_Slot5_I".CH05,
                   fOffset := 0.0,
                   sTag := "DB_Valves".HBL_HCV_616.Stat.Position,
                   fEngValue => #fDummy);
END_REGION

REGION Network 69: HBL_PT_618 HP Receiver pressure
   "fcAnalogInput"(bValidData := "RIO2_Slot5_I".CH06_ok,
                   iAI := "RIO2_Slot5_I".CH06,
                   fOffset := "DB_System".BarometricOffset,
                   sTag := "DB_AI".HBL_PT_618,
                   fEngValue => #fDummy);
END_REGION

REGION Network 70: HBL_CT_620 Gas detector recuperator popoff
   "fcAnalogInput"(bValidData := "RIO2_Slot5_I".CH07_ok,
                   iAI := "RIO2_Slot5_I".CH07,
                   fOffset := 0.0,
                   sTag := "DB_AI".HBL_CT_620,
                   fEngValue => #fDummy);
END_REGION

REGION Network 71: HBL_PT_635 Oil separator stage 1 oil return pressure
   "fcAnalogInput"(bValidData := false,
                   iAI := 0,
                   fOffset := "DB_System".BarometricOffset,
                   sTag := "DB_AI".HBL_PT_635,
                   fEngValue => #fDummy);
END_REGION

REGION Network 72: HBL_PT_636 Oil separator stage 2 oil return pressure
   "fcAnalogInput"(bValidData := false,
                   iAI := 0,
                   fOffset := "DB_System".BarometricOffset,
                   sTag := "DB_AI".HBL_PT_636,
                   fEngValue => #fDummy);
END_REGION

REGION Network 73: HBL_CT_643 Gas detector suction accumulator popoff
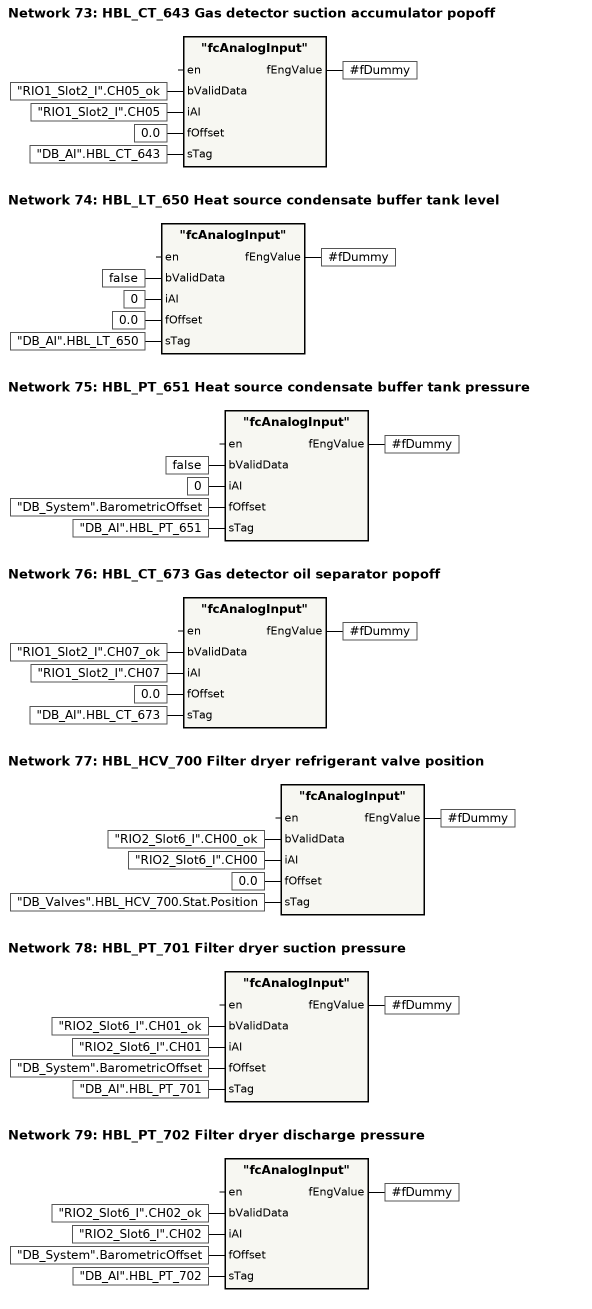
   "fcAnalogInput"(bValidData := "RIO1_Slot2_I".CH05_ok,
                   iAI := "RIO1_Slot2_I".CH05,
                   fOffset := 0.0,
                   sTag := "DB_AI".HBL_CT_643,
                   fEngValue => #fDummy);
END_REGION

REGION Network 74: HBL_LT_650 Heat source condensate buffer tank level
   "fcAnalogInput"(bValidData := false,
                   iAI := 0,
                   fOffset := 0.0,
                   sTag := "DB_AI".HBL_LT_650,
                   fEngValue => #fDummy);
END_REGION

REGION Network 75: HBL_PT_651 Heat source condensate buffer tank pressure
   "fcAnalogInput"(bValidData := false,
                   iAI := 0,
                   fOffset := "DB_System".BarometricOffset,
                   sTag := "DB_AI".HBL_PT_651,
                   fEngValue => #fDummy);
END_REGION

REGION Network 76: HBL_CT_673 Gas detector oil separator popoff
   "fcAnalogInput"(bValidData := "RIO1_Slot2_I".CH07_ok,
                   iAI := "RIO1_Slot2_I".CH07,
                   fOffset := 0.0,
                   sTag := "DB_AI".HBL_CT_673,
                   fEngValue => #fDummy);
END_REGION

REGION Network 77: HBL_HCV_700 Filter dryer refrigerant valve position
   "fcAnalogInput"(bValidData := "RIO2_Slot6_I".CH00_ok,
                   iAI := "RIO2_Slot6_I".CH00,
                   fOffset := 0.0,
                   sTag := "DB_Valves".HBL_HCV_700.Stat.Position,
                   fEngValue => #fDummy);
END_REGION

REGION Network 78: HBL_PT_701 Filter dryer suction pressure
   "fcAnalogInput"(bValidData := "RIO2_Slot6_I".CH01_ok,
                   iAI := "RIO2_Slot6_I".CH01,
                   fOffset := "DB_System".BarometricOffset,
                   sTag := "DB_AI".HBL_PT_701,
                   fEngValue => #fDummy);
END_REGION

REGION Network 79: HBL_PT_702 Filter dryer discharge pressure
   "fcAnalogInput"(bValidData := "RIO2_Slot6_I".CH02_ok,
                   iAI := "RIO2_Slot6_I".CH02,
                   fOffset := "DB_System".BarometricOffset,
                   sTag := "DB_AI".HBL_PT_702,
                   fEngValue => #fDummy);
END_REGION

REGION Network 80: HBL_PT_703 Filter dryer differential pressure
   // PT703 = PT701 - PT702 (Pressure drop)
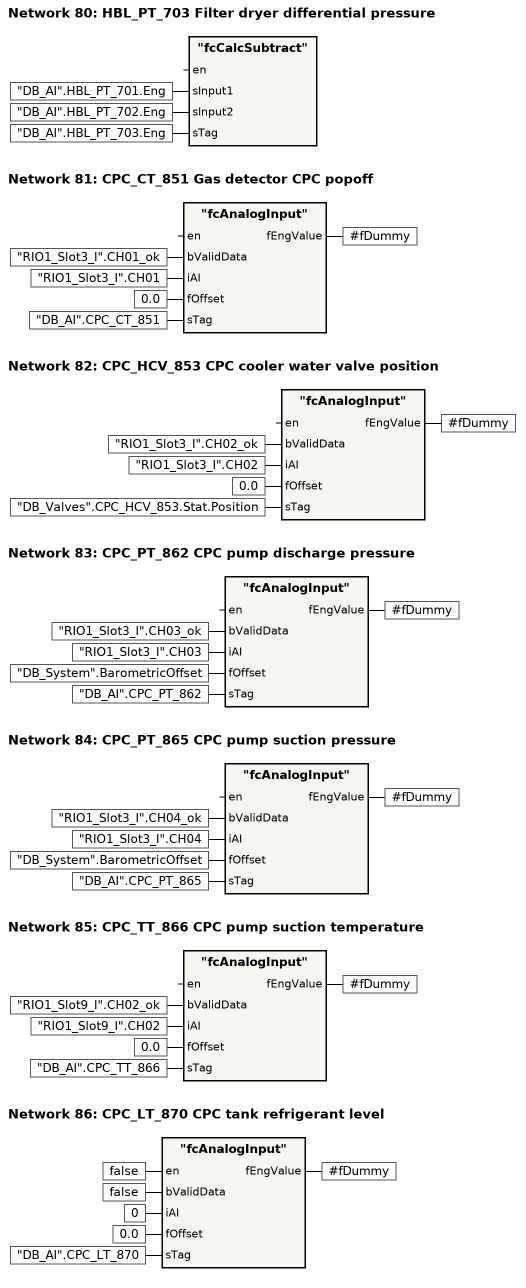
   "fcCalcSubtract"(sInput1 := "DB_AI".HBL_PT_701.Eng,
                    sInput2 := "DB_AI".HBL_PT_702.Eng,
                    sTag := "DB_AI".HBL_PT_703.Eng);
END_REGION

REGION Network 81: CPC_CT_851 Gas detector CPC popoff
   "fcAnalogInput"(bValidData := "RIO1_Slot3_I".CH01_ok,
                   iAI := "RIO1_Slot3_I".CH01,
                   fOffset := 0.0,
                   sTag := "DB_AI".CPC_CT_851,
                   fEngValue => #fDummy);
END_REGION

REGION Network 82: CPC_HCV_853 CPC cooler water valve position
   "fcAnalogInput"(bValidData := "RIO1_Slot3_I".CH02_ok,
                   iAI := "RIO1_Slot3_I".CH02,
                   fOffset := 0.0,
                   sTag := "DB_Valves".CPC_HCV_853.Stat.Position,
                   fEngValue => #fDummy);
END_REGION

REGION Network 83: CPC_PT_862 CPC pump discharge pressure
   "fcAnalogInput"(bValidData := "RIO1_Slot3_I".CH03_ok,
                   iAI := "RIO1_Slot3_I".CH03,
                   fOffset := "DB_System".BarometricOffset,
                   sTag := "DB_AI".CPC_PT_862,
                   fEngValue => #fDummy);
END_REGION

REGION Network 84: CPC_PT_865 CPC pump suction pressure
   "fcAnalogInput"(bValidData := "RIO1_Slot3_I".CH04_ok,
                   iAI := "RIO1_Slot3_I".CH04,
                   fOffset := "DB_System".BarometricOffset,
                   sTag := "DB_AI".CPC_PT_865,
                   fEngValue => #fDummy);
END_REGION

REGION Network 85: CPC_TT_866 CPC pump suction temperature
   "fcAnalogInput"(bValidData := "RIO1_Slot9_I".CH02_ok,
                   iAI := "RIO1_Slot9_I".CH02,
                   fOffset := 0.0,
                   sTag := "DB_AI".CPC_TT_866,
                   fEngValue => #fDummy);
END_REGION

REGION Network 86: CPC_LT_870 CPC tank refrigerant level
   IF false THEN
       "fcAnalogInput"(bValidData := false,
                       iAI := 0,
                       fOffset := 0.0,
                       sTag := "DB_AI".CPC_LT_870,
                       fEngValue => #fDummy);
   END_IF;
END_REGION

REGION Network 87: CPC_TT_871 CPC tank refrigerant temperature
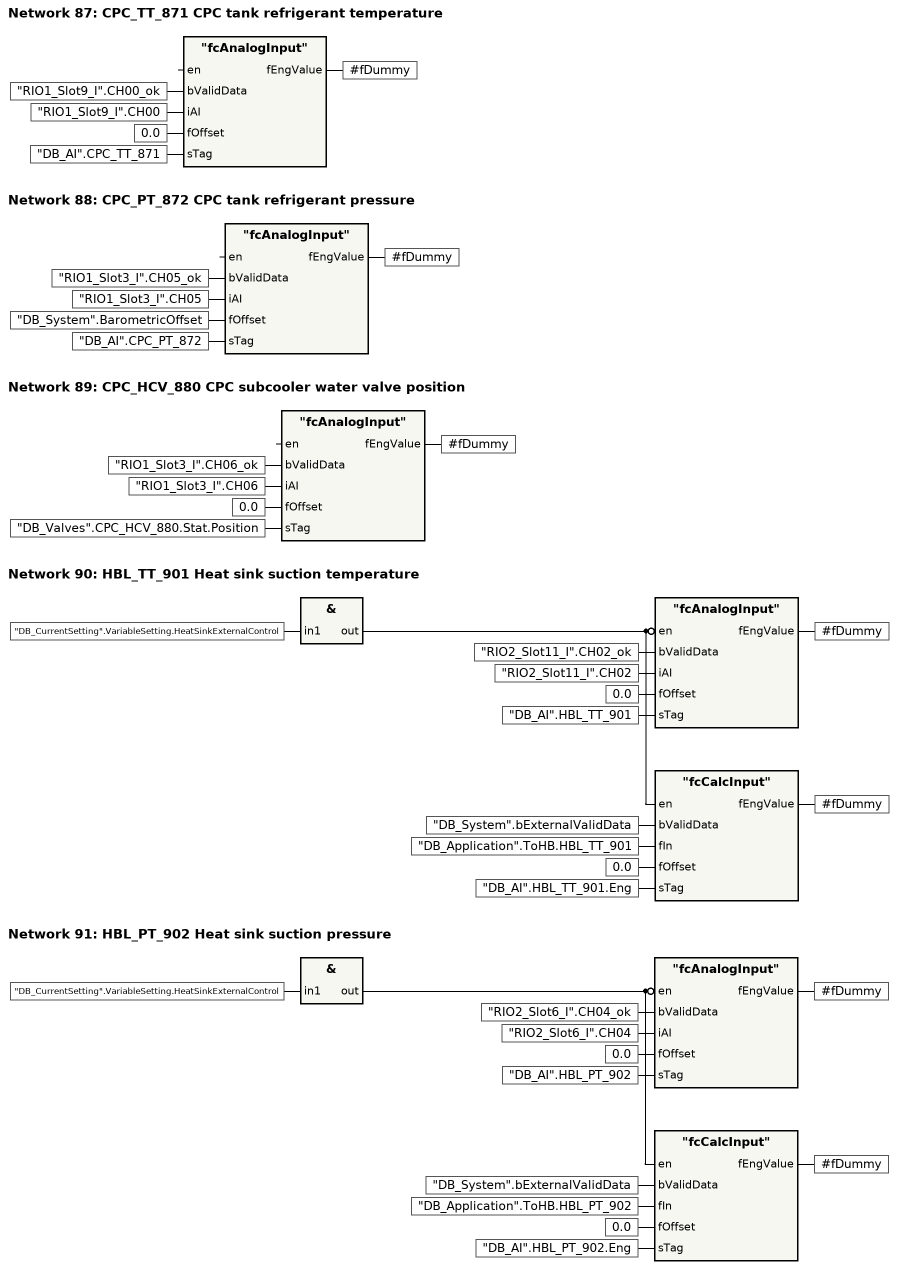
   "fcAnalogInput"(bValidData := "RIO1_Slot9_I".CH00_ok,
                   iAI := "RIO1_Slot9_I".CH00,
                   fOffset := 0.0,
                   sTag := "DB_AI".CPC_TT_871,
                   fEngValue => #fDummy);
END_REGION

REGION Network 88: CPC_PT_872 CPC tank refrigerant pressure
   "fcAnalogInput"(bValidData := "RIO1_Slot3_I".CH05_ok,
                   iAI := "RIO1_Slot3_I".CH05,
                   fOffset := "DB_System".BarometricOffset,
                   sTag := "DB_AI".CPC_PT_872,
                   fEngValue => #fDummy);
END_REGION

REGION Network 89: CPC_HCV_880 CPC subcooler water valve position
   "fcAnalogInput"(bValidData := "RIO1_Slot3_I".CH06_ok,
                   iAI := "RIO1_Slot3_I".CH06,
                   fOffset := 0.0,
                   sTag := "DB_Valves".CPC_HCV_880.Stat.Position,
                   fEngValue => #fDummy);
END_REGION

REGION Network 90: HBL_TT_901 Heat sink suction temperature
   #_w1 := "DB_CurrentSetting".VariableSetting.HeatSinkExternalControl;
   IF NOT "DB_CurrentSetting".VariableSetting.HeatSinkExternalControl THEN
       "fcAnalogInput"(bValidData := "RIO2_Slot11_I".CH02_ok,
                       iAI := "RIO2_Slot11_I".CH02,
                       fOffset := 0.0,
                       sTag := "DB_AI".HBL_TT_901,
                       fEngValue => #fDummy);
   END_IF;
   IF #_w1 THEN
       "fcCalcInput"(bValidData := "DB_System".bExternalValidData,
                     fIn := "DB_Application".ToHB.HBL_TT_901,
                     fOffset := 0.0,
                     sTag := "DB_AI".HBL_TT_901.Eng,
                     fEngValue => #fDummy);
   END_IF;
END_REGION

REGION Network 91: HBL_PT_902 Heat sink suction pressure
   #_w1 := "DB_CurrentSetting".VariableSetting.HeatSinkExternalControl;
   IF NOT "DB_CurrentSetting".VariableSetting.HeatSinkExternalControl THEN
       "fcAnalogInput"(bValidData := "RIO2_Slot6_I".CH04_ok,
                       iAI := "RIO2_Slot6_I".CH04,
                       fOffset := 0.0,
                       sTag := "DB_AI".HBL_PT_902,
                       fEngValue => #fDummy);
   END_IF;
   IF #_w1 THEN
       "fcCalcInput"(bValidData := "DB_System".bExternalValidData,
                     fIn := "DB_Application".ToHB.HBL_PT_902,
                     fOffset := 0.0,
                     sTag := "DB_AI".HBL_PT_902.Eng,
                     fEngValue => #fDummy);
   END_IF;
END_REGION

REGION Network 92: HBL_CT_950 Gas detector container/compressor room
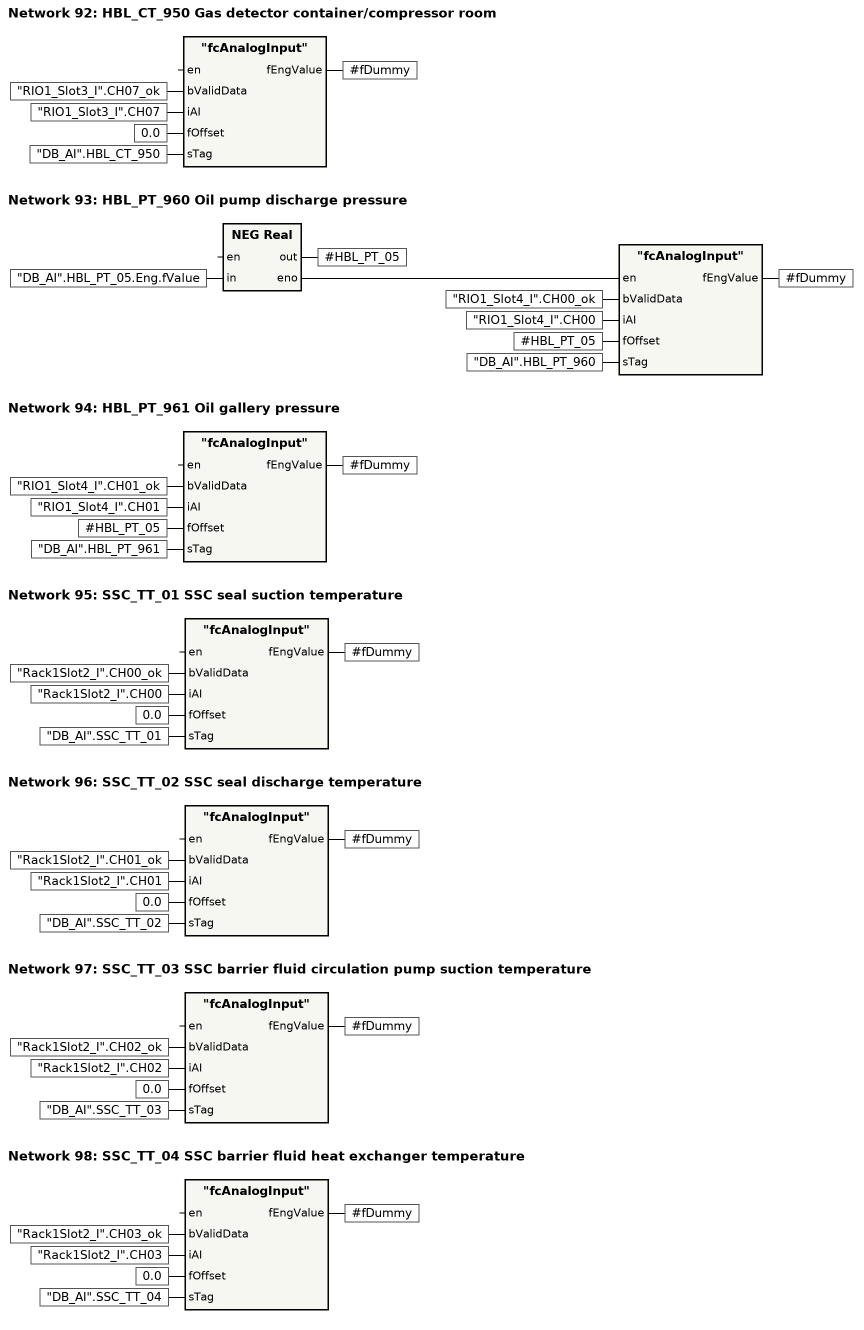
   "fcAnalogInput"(bValidData := "RIO1_Slot3_I".CH07_ok,
                   iAI := "RIO1_Slot3_I".CH07,
                   fOffset := 0.0,
                   sTag := "DB_AI".HBL_CT_950,
                   fEngValue => #fDummy);
END_REGION

REGION Network 93: HBL_PT_960 Oil pump discharge pressure
   // Relative to the crankcase pressure
   #HBL_PT_05 := -"DB_AI".HBL_PT_05.Eng.fValue;
   "fcAnalogInput"(bValidData := "RIO1_Slot4_I".CH00_ok,
                   iAI := "RIO1_Slot4_I".CH00,
                   fOffset := #HBL_PT_05,
                   sTag := "DB_AI".HBL_PT_960,
                   fEngValue => #fDummy);
END_REGION

REGION Network 94: HBL_PT_961 Oil gallery pressure
   // Relative to the crankcase pressure
   "fcAnalogInput"(bValidData := "RIO1_Slot4_I".CH01_ok,
                   iAI := "RIO1_Slot4_I".CH01,
                   fOffset := #HBL_PT_05,
                   sTag := "DB_AI".HBL_PT_961,
                   fEngValue => #fDummy);
END_REGION

REGION Network 95: SSC_TT_01 SSC seal suction temperature
   "fcAnalogInput"(bValidData := "Rack1Slot2_I".CH00_ok,
                   iAI := "Rack1Slot2_I".CH00,
                   fOffset := 0.0,
                   sTag := "DB_AI".SSC_TT_01,
                   fEngValue => #fDummy);
END_REGION

REGION Network 96: SSC_TT_02 SSC seal discharge temperature
   "fcAnalogInput"(bValidData := "Rack1Slot2_I".CH01_ok,
                   iAI := "Rack1Slot2_I".CH01,
                   fOffset := 0.0,
                   sTag := "DB_AI".SSC_TT_02,
                   fEngValue => #fDummy);
END_REGION

REGION Network 97: SSC_TT_03 SSC barrier fluid circulation pump suction temperature
   "fcAnalogInput"(bValidData := "Rack1Slot2_I".CH02_ok,
                   iAI := "Rack1Slot2_I".CH02,
                   fOffset := 0.0,
                   sTag := "DB_AI".SSC_TT_03,
                   fEngValue => #fDummy);
END_REGION

REGION Network 98: SSC_TT_04 SSC barrier fluid heat exchanger temperature
   "fcAnalogInput"(bValidData := "Rack1Slot2_I".CH03_ok,
                   iAI := "Rack1Slot2_I".CH03,
                   fOffset := 0.0,
                   sTag := "DB_AI".SSC_TT_04,
                   fEngValue => #fDummy);
END_REGION

REGION Network 99: SSC_PIT_01 SSC barrier fluid accumulator pressure
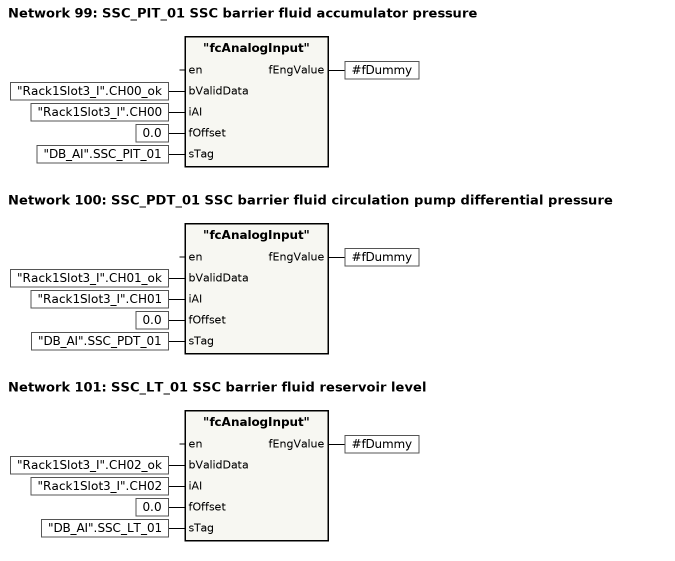
   "fcAnalogInput"(bValidData := "Rack1Slot3_I".CH00_ok,
                   iAI := "Rack1Slot3_I".CH00,
                   fOffset := 0.0,
                   sTag := "DB_AI".SSC_PIT_01,
                   fEngValue => #fDummy);
END_REGION

REGION Network 100: SSC_PDT_01 SSC barrier fluid circulation pump differential pressure
   "fcAnalogInput"(bValidData := "Rack1Slot3_I".CH01_ok,
                   iAI := "Rack1Slot3_I".CH01,
                   fOffset := 0.0,
                   sTag := "DB_AI".SSC_PDT_01,
                   fEngValue => #fDummy);
END_REGION

REGION Network 101: SSC_LT_01 SSC barrier fluid reservoir level
   "fcAnalogInput"(bValidData := "Rack1Slot3_I".CH02_ok,
                   iAI := "Rack1Slot3_I".CH02,
                   fOffset := 0.0,
                   sTag := "DB_AI".SSC_LT_01,
                   fEngValue => #fDummy);
END_REGION
END_FUNCTION_BLOCK

FUNCTION "fcCalcInput" : Void
{ S7_Optimized_Access := 'TRUE' }
AUTHOR : Heaten
VERSION : 0.1
   VAR_INPUT 
      bValidData : Bool;
      fIn : Real;
      fOffset : Real;
   END_VAR

   VAR_OUTPUT 
      fEngValue : Real;
   END_VAR

   VAR_IN_OUT 
      sTag : "stCalcValue";
   END_VAR

   VAR_TEMP 
      fSlope : Real;
      fIntercept : Real;
      fValue : Real;
   END_VAR


BEGIN
	// Take an already-scaled value and convert it to a Calc value
	// Difference over fcCalcAssign is that it has a bottom value, and allows adding an offset
	
	// Scaling
	IF NOT #bValidData OR "isNaN"(#fValue) THEN
	    // Error value
	    #sTag.bError := TRUE;
	    #sTag.fValue := "NaN"();
	    #sTag.bLimited := FALSE;
	ELSE
	    #sTag.bError := FALSE;
	    #fValue := #fIn + #fOffset;
	    // Apply limiting, if enabled
	    "fcCalcAssign"(fValue := #fValue, sTag := #sTag);
	END_IF;
	
	// Local output
	#fEngValue := #sTag.#fValue;
	
END_FUNCTION

FUNCTION "fcCalcSubtract" : Void
{ S7_Optimized_Access := 'TRUE' }
VERSION : 0.1
   VAR_INPUT 
      sInput1 : "stCalcValue";
      sInput2 : "stCalcValue";
   END_VAR

   VAR_IN_OUT 
      sTag : "stCalcValue";
   END_VAR

   VAR_TEMP 
      fResult : Real;
   END_VAR


BEGIN
	// Subtract two Calc values
	// A subtraction is not defined if either or both arguments are not defined, or more directly:
	// If one or both values is #NaN, the result should always be #NaN.
	
	IF #sInput1.bError = TRUE OR #sInput2.bError = TRUE OR "isNaN"(In := #sInput1.fValue) OR "isNaN"(In := #sInput2.fValue) THEN
	    #sTag.bError := TRUE;
	    #sTag.fValue := "NaN"();
	ELSE
	    #sTag.bError := FALSE;
	    // Do the subtraction
	    #fResult := #sInput1.fValue - #sInput2.fValue;
	    // Handle limiting
	    "fcCalcAssign"(fValue := #fResult, sTag := #sTag);
	END_IF;
	
	
END_FUNCTION

FUNCTION_BLOCK "InverterDriveProcessing"   // FB12, FBD
TITLE = Inverter drive processing
{ S7_Optimized_Access := 'FALSE' }
AUTHOR : Heaten
VERSION : 0.1
// Command and status
// stored: AutoNumber true, IsIECCheckEnabled false, SetENOAutomatically false, UDAEnableTagReadback false
   VAR
      HBL_SC_02 { ExternalAccessible := 'False'; ExternalVisible := 'False'; ExternalWritable := 'False'} : "fbACS880";
      HBL_SC_03 { S7_SetPoint := 'True'} : "fbACS880";
      HBL_SC_01 { ExternalAccessible := 'False'; ExternalVisible := 'False'; ExternalWritable := 'False'} : "fbACS880";
      HBL_SC_10 { ExternalAccessible := 'False'; ExternalVisible := 'False'; ExternalWritable := 'False'} : "fbACS880";
   END_VAR
   VAR DB_SPECIFIC
      State : Array[0..7] of Bool;   // Profinet online state (1 bit per node)
      RetVal { ExternalAccessible := 'False'; ExternalVisible := 'False'; ExternalWritable := 'False'} : Int;   // Error code internal to DeviceStates
   END_VAR
BEGIN

REGION Network 1: Comm status all Profinet devices
   // Mode 1 = IO devices are configured
   // Mode 2 = IO devices are faulty
   // Mode 3 = IO devices are disabled
   // Mode 4 = IO devices exist
   // Mode 5 = IO devices for which a problem has occurred
   // online state bit corresponds to "Profinet device number" -> CHECK THIS IN DEVICE CONFIGURATION
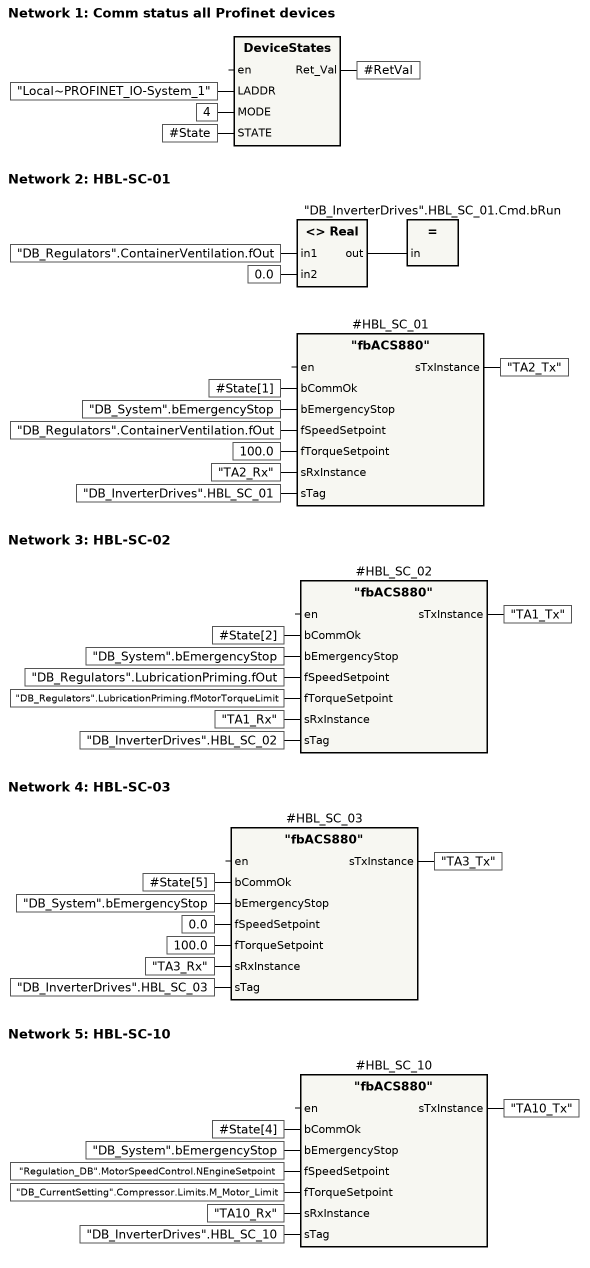
   #RetVal := DeviceStates(LADDR := "Local~PROFINET_IO-System_1", MODE := 4, STATE := #State);
END_REGION

REGION Network 2: HBL-SC-01
   "DB_InverterDrives".HBL_SC_01.Cmd.bRun := "DB_Regulators".ContainerVentilation.fOut <> 0.0;
   #HBL_SC_01(bCommOk := #State[1],   // "fbACS880"
              bEmergencyStop := "DB_System".bEmergencyStop,
              fSpeedSetpoint := "DB_Regulators".ContainerVentilation.fOut,
              fTorqueSetpoint := 100.0,
              sRxInstance := "TA2_Rx",
              sTag := "DB_InverterDrives".HBL_SC_01,
              sTxInstance => "TA2_Tx");
END_REGION

REGION Network 3: HBL-SC-02
   #HBL_SC_02(bCommOk := #State[2],   // "fbACS880"
              bEmergencyStop := "DB_System".bEmergencyStop,
              fSpeedSetpoint := "DB_Regulators".LubricationPriming.fOut,
              fTorqueSetpoint := "DB_Regulators".LubricationPriming.fMotorTorqueLimit,
              sRxInstance := "TA1_Rx",
              sTag := "DB_InverterDrives".HBL_SC_02,
              sTxInstance => "TA1_Tx");
END_REGION

REGION Network 4: HBL-SC-03
   #HBL_SC_03(bCommOk := #State[5],   // "fbACS880"
              bEmergencyStop := "DB_System".bEmergencyStop,
              fSpeedSetpoint := 0.0,
              fTorqueSetpoint := 100.0,
              sRxInstance := "TA3_Rx",
              sTag := "DB_InverterDrives".HBL_SC_03,
              sTxInstance => "TA3_Tx");
END_REGION

REGION Network 5: HBL-SC-10
   #HBL_SC_10(bCommOk := #State[4],   // "fbACS880"
              bEmergencyStop := "DB_System".bEmergencyStop,
              fSpeedSetpoint := "Regulation_DB".MotorSpeedControl.NEngineSetpoint,
              fTorqueSetpoint := "DB_CurrentSetting".Compressor.Limits.M_Motor_Limit,
              sRxInstance := "TA10_Rx",
              sTag := "DB_InverterDrives".HBL_SC_10,
              sTxInstance => "TA10_Tx");
END_REGION
END_FUNCTION_BLOCK

FUNCTION_BLOCK "fbACS880"   // FB22, FBD
TITLE = Interface block for ABB ACS880
{ S7_Optimized_Access := 'TRUE' }
AUTHOR : Heaten
VERSION : 0.1
// stored: AutoNumber true, IsIECCheckEnabled false, IsRetainMemResEnabled false, MemoryReserve 0, SetENOAutomatically false, UDAEnableTagReadback false
   VAR_INPUT
      bCommOk : Bool;   // 0 = comm fail
      bEmergencyStop : Bool;   // 1 = E-stop, 0 = ok
      fSpeedSetpoint : Real;   // rpm
      fTorqueSetpoint : Real;   // %
      sRxInstance : "stABB_ACSx80_Rx";   // Input data raw
   END_VAR
   VAR_OUTPUT
      sTxInstance : "stABB_ACSx80_Tx";   // Output data raw
   END_VAR
   VAR_IN_OUT
      sTag : "stInverterDrive";   // This drive
   END_VAR
   VAR
      ResetTimer : TP_TIME;   // NB: Pulse timer!
   END_VAR
   VAR_TEMP
      Dummy : Real;
      Speed : Int;
      Torque : Int;
   END_VAR
BEGIN

REGION Network 1: Fieldbus comm ok
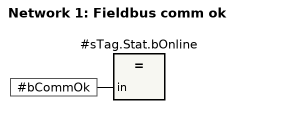
   #sTag.Stat.bOnline := #bCommOk;
END_REGION

REGION Network 2 (SCL): Data processing: READ
   // handle Act1 & Act2
   "fcAnalogInput"(bValidData := #bCommOk, iAI := WORD_TO_INT(#sRxInstance.Act1), fOffset := 0.0, sTag := #sTag.Stat.Speed, fEngValue => #Dummy);
   "fcAnalogInput"(bValidData := #bCommOk, iAI := WORD_TO_INT(#sRxInstance.Act2), fOffset := 0.0, sTag := #sTag.Stat.Torque, fEngValue => #Dummy);
   "fcAnalogInput"(bValidData := #bCommOk, iAI := WORD_TO_INT(#sRxInstance.DataIO_12), fOffset := 0.0, sTag := #sTag.Stat.Power, fEngValue => #Dummy);

   // Status Word
   IF #bCommOk = FALSE THEN
       // Zero out all data on comm error
       #sTag.Stat.bRemote := FALSE;
       #sTag.Stat.bRun := FALSE;
       #sTag.Stat.bTrip := FALSE;
       #sTag.Stat.bReady := FALSE;
   ELSE
       // Status Word (ABB Drives profile)
       // BIT  NAME            STATE
       // 0    RDY_ON          Ready to Switch On
       // 1    RDY_RUN         0 = OFF1 active, 1 = Ready to operate
       // 2    RDY_REF         Operation enabled
       // 3    TRIPPED         Fault
       // 4    OFF_2_STATUS    0 = OFF2 active, 1 = OFF2 inactive
       // 5    OFF_3_STATUS    0 = OFF3 active, 1 = OFF3 inactive
       // 6    SWC_ON_INHIB    1 = Switch-on inhibited
       // 7    ALARM           0 = No warning/alarm, 1 = warning/alarm
       // 8    AT_SETPOINT     1 = actual value within tolerance of Ref
       // 9    REMOTE          0 = local control 1 = remote control
       // 10   ABOVE_LIMIT     1 = actual speed >= supervision limit
       // 11   USER_0          
       // 12   USER_1
       // 13   USER_2
       // 14   USER_3
       // 15   Reserved by ABB
       #sTag.Stat.bReady := #sRxInstance.SW.%X0;
       #sTag.Stat.bRun := #sRxInstance.SW.%X2;
       #sTag.Stat.bTrip := #sRxInstance.SW.%X3;
       #sTag.Stat.bRemote := #sRxInstance.SW.%X9;

       // Further optional processing based on variant
       CASE #sTag.nVariant OF
           0 : ;
           1 : ;
       END_CASE;
   END_IF;
END_REGION

REGION Network 3 (SCL): Data processing: WRITE
   // Outputs get written even if there is comm error
   // Control Word (ABB Drives profile)
   // BIT  NAME            STATE
   // 0    OFF1_CONTROL    0 = OFF1 Active, 1 = Proceed to READY TO OPERATE
   // 1    OFF2_CONTROL    0 = OFF2 Active, 1 = Continue operation
   // 2    OFF3_CONTROL    0 = OFF3 Active, 1 = Continue operation
   // 3    INHIBIT_OPERATION 0 = inhibit, 1 = Proceed to OPERATION ENABLED (Run?)
   // 4    RAMP_OUT_ZERO   0 = force ramp output to zero, 1 = normal operation
   // 5    RAMP_HOLD       0 = halt ramping (hold output), 1 = normal operation
   // 6    RAMP_IN_ZERO    0 = force ramp input to zero, 1 = normal operation
   // 7    RESET           0 = normal operation, 1 = reset fault
   // 8    JOGGING_1       0 = normal operation, 1 = run at Jogging 1 speed
   // 9    JOGGING_2       0 = normal operation, 1 = run at Jogging 2 speed
   // 10   REMOTE_CMD      0 = ?, 1 = fieldbus controlled
   // 11   EXT_CTRL_LOC    0 = EXT1, 1 = EXT2
   // 12   USER_0
   // 13   USER_1
   // 14   USER_2
   // 15   USER_3
   // NOTE: the firmware manual describes a state machine for starting the drive. But the transitions from
   // one state to another are levels and not edges, therefore several conditions can be combined and sent
   // at the same time.
   // Stop : CW = 16#0476
   // Ready : CW = 16#47E
   // Run  : CW = 16#047F
   // Reset: CW = 16#04F6
   // NOTE 2: sTag.Cmd.bReady is for enabling the drive without running it; sTag.Cmd.bRun will override this, so don't use bReady to turn the drive on and off

   // Make reset a pulse
   #ResetTimer(IN := #sTag.Cmd.bReset, PT := T#3s);

   // Control word
   IF #bEmergencyStop = TRUE THEN
       #sTxInstance.CW := 16#0476;
   ELSIF #ResetTimer.Q THEN
       #sTxInstance.CW := 16#04F6;
       #sTag.Cmd.bReset := FALSE;
   ELSIF #sTag.Cmd.bManualRun = TRUE AND #sTag.Cmd.bManualMode = TRUE THEN
       #sTxInstance.CW := 16#047F;
   ELSIF #sTag.Cmd.bRun = TRUE THEN
       #sTxInstance.CW := 16#047F;
   ELSIF #sTag.Cmd.bReady = TRUE THEN
       #sTxInstance.CW := 16#047E;
   ELSE
       #sTxInstance.CW := 16#0476;
   END_IF;

   // Setpoints
   IF #bEmergencyStop = TRUE THEN
       "fcCalcAssign"(fValue := 0.0, sTag := #sTag.Cmd.Speed.Eng);
       "fcCalcAssign"(fValue := 0.0, sTag := #sTag.Cmd.Torque.Eng);
       #sTag.Cmd.bManualMode := FALSE;
       #sTag.Cmd.fManualSpeed := 0.0;
   ELSIF #sTag.Cmd.bManualMode = TRUE THEN
       "fcCalcAssign"(fValue := #sTag.Cmd.fManualSpeed, sTag:= #sTag.Cmd.Speed.Eng);
       "fcCalcAssign"(fValue := #sTag.Cmd.fManualTorque, sTag := #sTag.Cmd.Torque.Eng);
   ELSE
       // Allow Manual Mode to take over from auto in run state and with same setpoints
       IF #sTag.Stat.bRun = TRUE THEN
           #sTag.Cmd.bManualRun := #sTag.Cmd.bRun;
           #sTag.Cmd.fManualSpeed := #sTag.Cmd.Speed.Eng.fValue;
           #sTag.Cmd.fManualTorque := #sTag.Cmd.Torque.Eng.fValue;
       END_IF;

       "fcCalcAssign"(fValue := #fSpeedSetpoint, sTag:= #sTag.Cmd.Speed.Eng);
       "fcCalcAssign"(fValue := #fTorqueSetpoint, sTag := #sTag.Cmd.Torque.Eng);
   END_IF;

   // Write to fieldbus
   "fcAnalogOutput"(bOutputOk := #bCommOk, sTag := #sTag.Cmd.Speed, iAO => #Speed);
   "fcAnalogOutput"(bOutputOk := #bCommOk, sTag := #sTag.Cmd.Torque, iAO => #Torque);

   #sTxInstance.Ref1 := INT_TO_WORD(#Speed);
   #sTxInstance.Ref2 := INT_TO_WORD(#Torque);
END_REGION
END_FUNCTION_BLOCK

FUNCTION_BLOCK "fbProcessValve2_V2"   // FB67, FBD
TITLE = Process valve control
{ S7_Optimized_Access := 'TRUE' }
AUTHOR : Heaten
VERSION : 1.0
// stored: AutoNumber true, IsIECCheckEnabled false, IsRetainMemResEnabled false, MemoryReserve 0, SetENOAutomatically false, UDAEnableTagReadback false
   VAR_INPUT
      bOpenReq : Bool;   // 1 = open valve, 0 = do not open valve (Level signal)
      bCloseReq : Bool;   // 1 = close valve, 0 = do not close valve (Level signal)
      bOpenStat : Bool;   // 1 = valve is open, 0 = valve is not open
      bClosedStat : Bool;   // 1 = valve is closed, 0 = valve is not closed
   END_VAR
   VAR_OUTPUT
      bOpenCmd : Bool;
      bCloseCmd : Bool;
   END_VAR
   VAR_IN_OUT
      sTag : "stProcessValve2";
   END_VAR
   VAR
      OpenTimer : TON_TIME;
      CloseTimer { S7_SetPoint := 'True'} : TON_TIME;
   END_VAR
   VAR_TEMP
      Opening : Bool;
      Closing : Bool;
      OpenError : Bool;
      CloseError : Bool;
      OpenReq : Bool;
      CloseReq : Bool;
   END_VAR
   VAR CONSTANT
      STATE_UNKNOWN : USInt := 0;
      STATE_CLOSED : USInt := 1;
      STATE_OPEN : USInt := 2;
      STATE_CLOSING : USInt := 3;
      STATE_OPENING : USInt := 4;
      STATE_CLOSE_ERROR : USInt := 5;
      STATE_OPEN_ERROR : USInt := 6;
   END_VAR
BEGIN

REGION Network 1 (SCL): Description & version history
   // Remember to update the version in the block properties!
   // Process valve control with decoupled states
   // - valve state is directly represented by the feedback
   // - requests are level signals
   // - valve commands are conditions and not states
   // - errors are conditions and not states
   // - different concerns are decoupled: valve state, request & command, error detection
   // - needs no initial state detection or special handling if valve position feedback disappears

   // V1.0.0.0 08.03.2025 HEATEN
   // - Initial version
END_REGION

REGION Network 2: Open Request
   // Choose between auto & manual
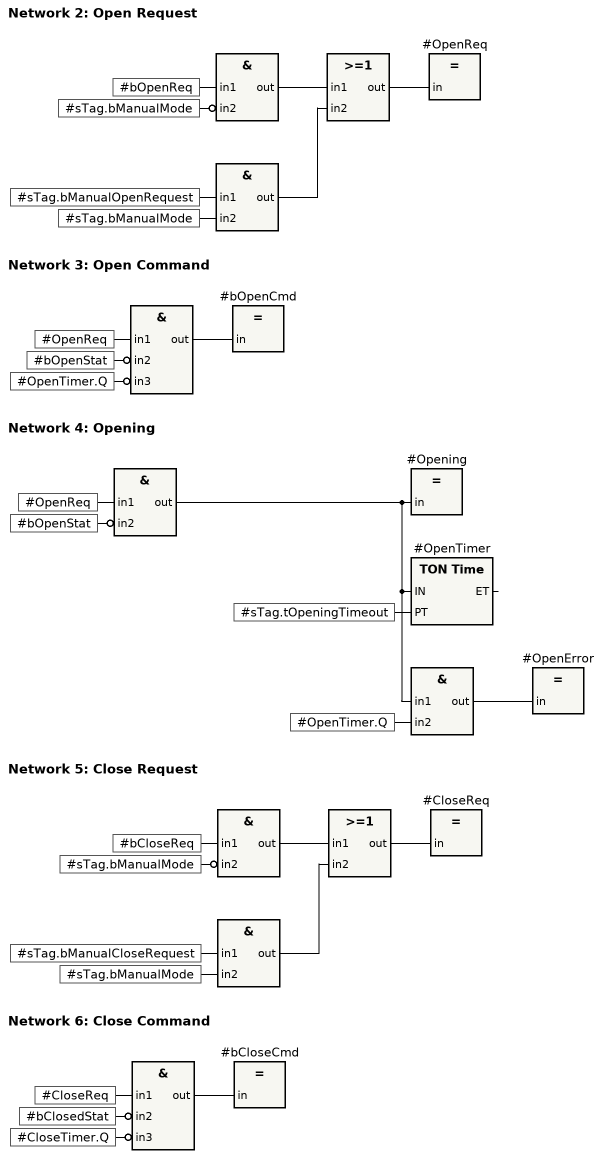
   #OpenReq := (#bOpenReq AND NOT #sTag.bManualMode) OR (#sTag.bManualOpenRequest AND #sTag.bManualMode);
END_REGION

REGION Network 3: Open Command
   // Send the command when the request to open is given
   // Stop when the open status is received or timoeut has occurred
   #bOpenCmd := #OpenReq AND NOT #bOpenStat AND NOT #OpenTimer.Q;
END_REGION

REGION Network 4: Opening
   // Opening as long as the open request is given and no open status received
   // Open timer fires when the request to open doesn't result in an open status after the timeout period
   // Open error active when opening and timeout occurs. Clears when the request is withdrawn or open status received
   #Opening := #OpenReq AND NOT #bOpenStat;
   #OpenTimer(IN := #Opening, PT := #sTag.tOpeningTimeout);   // TON
   #OpenError := #Opening AND #OpenTimer.Q;
END_REGION

REGION Network 5: Close Request
   // Choose between auto & manual
   #CloseReq := (#bCloseReq AND NOT #sTag.bManualMode) OR (#sTag.bManualCloseRequest AND #sTag.bManualMode);
END_REGION

REGION Network 6: Close Command
   // Send the command when the request to close is given
   // Stop when the closed status is received or timoeut has occurred
   #bCloseCmd := #CloseReq AND NOT #bClosedStat AND NOT #CloseTimer.Q;
END_REGION

REGION Network 7: Closing
   // Closing as long as the close request is given and no closed status received
   // Close Timer fires when the request to close doesn't result in a closed status after the timeout period
   // Close error active when closing and timeout occurs. Clears when the request is withdrawn or closed status received
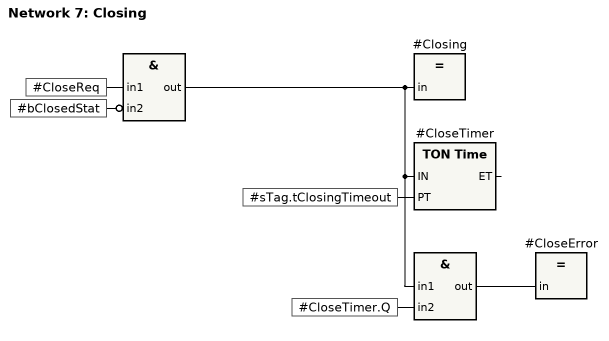
   #Closing := #CloseReq AND NOT #bClosedStat;
   #CloseTimer(IN := #Closing, PT := #sTag.tClosingTimeout);   // TON
   #CloseError := #Closing AND #CloseTimer.Q;
END_REGION

REGION Network 8 (SCL): State representation
   // The order is important, otherwise some conditions are never detected
   IF #OpenError = TRUE THEN
       #sTag.nState := #STATE_OPEN_ERROR;
   ELSIF #CloseError = TRUE THEN
       #sTag.nState := #STATE_CLOSE_ERROR;
   ELSIF #Opening = TRUE THEN
       #sTag.nState := #STATE_OPENING;
   ELSIF #Closing = TRUE THEN
       #sTag.nState := #STATE_CLOSING;
   ELSIF #bOpenStat = TRUE THEN
       #sTag.nState := #STATE_OPEN;
   ELSIF #bClosedStat = TRUE THEN
       #sTag.nState := #STATE_CLOSED;
   ELSE
       #sTag.nState := #STATE_UNKNOWN;
   END_IF;
END_REGION

REGION Network 9 (SCL): Mirror in HMI
   #sTag.bOpenRequest := #OpenReq;
   #sTag.bCloseRequest := #CloseReq;
   #sTag.bOpenStatus := #bOpenStat;
   #sTag.bClosedStatus := #bClosedStat;
   #sTag.bOpenCommand := #bOpenCmd;
   #sTag.bCloseCommand := #bCloseCmd;
END_REGION
END_FUNCTION_BLOCK

FUNCTION_BLOCK "Simulation"   // FB63, FBD
TITLE = Simulation of process values
{ S7_Optimized_Access := 'TRUE' }
AUTHOR : Heaten
VERSION : 0.1
// Simulate process values
// stored: AutoNumber true, IsIECCheckEnabled false, IsRetainMemResEnabled false, MemoryReserve 0, SetENOAutomatically false, UDAEnableTagReadback false
   VAR
      OilSump { S7_SetPoint := 'True'} : "fbButterworthLPF1";
      CPCPump { ExternalAccessible := 'False'; ExternalVisible := 'False'; ExternalWritable := 'False'; S7_SetPoint := 'True'} : "fbCPCPumpSim";
      HeatSource { S7_SetPoint := 'True'} : "fbButterworthLPF1";
   END_VAR
   VAR RETAIN
      fHeatSourceGain { S7_SetPoint := 'True'} : Real := 1.2;   // Conversion factor, % valve opening to HX temperature
   END_VAR
   VAR_TEMP
      fSumpHeatingTarget : Real;
      fOilSumpTemp : Real;
      fCPCDischarge : Real;
      fHeatSourceTarget : Real;
      fHeatSourceSimulated : Real;
   END_VAR
   VAR_TEMP   // added for the SCL form of the ladder/FBD networks
      _w1 : Bool;
   END_VAR
BEGIN

REGION Network 1 (SCL): Block comments
   // Don't put as comments under Block Title as this automatically appears in the weirdest places
   // A collection of hacks to provide feedback from the missing physical processes
END_REGION

REGION Network 2 (SCL): Simulation HBL-SC-10
   IF "DB_Alarms"."1110_HBL_SC_10_CommError".sState.bActive = TRUE THEN
       "DB_InverterDrives".HBL_SC_10.Stat.bOnline := TRUE;
       "DB_InverterDrives".HBL_SC_10.Stat.bReady := "DB_InverterDrives".HBL_SC_10.Cmd.bReady OR "DB_InverterDrives".HBL_SC_10.Cmd.bRun;
       "DB_InverterDrives".HBL_SC_10.Stat.bRemote := TRUE;
       "DB_InverterDrives".HBL_SC_10.Stat.bRun := "DB_InverterDrives".HBL_SC_10.Cmd.bRun;
       "DB_InverterDrives".HBL_SC_10.Stat.Speed.Eng.bError := FALSE;
       "DB_InverterDrives".HBL_SC_10.Stat.Speed.Eng.fValue :="DB_InverterDrives".HBL_SC_10.Cmd.Speed.Eng.fValue;
       "DB_InverterDrives".HBL_SC_10.Stat.Torque.Eng.bError := FALSE;
       "DB_InverterDrives".HBL_SC_10.Stat.Torque.Eng.fValue := "DB_InverterDrives".HBL_SC_10.Cmd.Torque.Eng.fValue;
       "DB_InverterDrives".HBL_SC_10.Stat.Power.Eng.bError := FALSE;
       "DB_InverterDrives".HBL_SC_10.Stat.Power.Eng.fValue := 355.0 * "DB_InverterDrives".HBL_SC_10.Stat.Speed.Eng.fValue/1500.0;
   END_IF;
END_REGION

REGION Network 3 (SCL): Simulation for oil gallery pressure
   // Just a rough hack to get some representative pressures
   // Oil pressure is always the sum of the two pumps. The primer pump will drop out above a certain oil pressure and come back on
   // We let the regulator decide for us and just do the sum
   // Primer pump: 100kPa at 5000rpm = 0.02 kPa/rpm (0.021747 to make it look more "random")
   // Main pump: 0.250 kPa/rpm to be above the minimum of 0.167 kPa/rpm to avoid warnings (0.257 to make it look more "random")
   // Filter deltaP = 20kPa
   "fcCalcAssign"(fValue := "DB_InverterDrives".HBL_SC_02.Stat.Speed.Eng.fValue * 0.021747 + "DB_InverterDrives".HBL_SC_10.Stat.Speed.Eng.fValue * 0.257,
                  sTag := "DB_AI".HBL_PT_960.Eng);
   "DB_AI".HBL_PT_961.Eng.bCheckLimits := TRUE;   // Limit to min & max
   "fcCalcAssign"(fValue := "DB_AI".HBL_PT_960.Eng.fValue - 20.0, sTag := "DB_AI".HBL_PT_961.Eng);
END_REGION

REGION Network 4: Simulation for Oil Sump Temperature
   // Thermal time constant: estimate 30 minutes to go from ambient to 45C
   // 5 tau = 30 minutes, or tau = 360 sec, or fc = 1/(2*pi*tau) = 0.00044210Hz (0.44mHz)
   // Go to 45C on Group 1 heaters, go to 82C on Group 1 + 2 heaters
   // When cooling, go towards the container air temperature
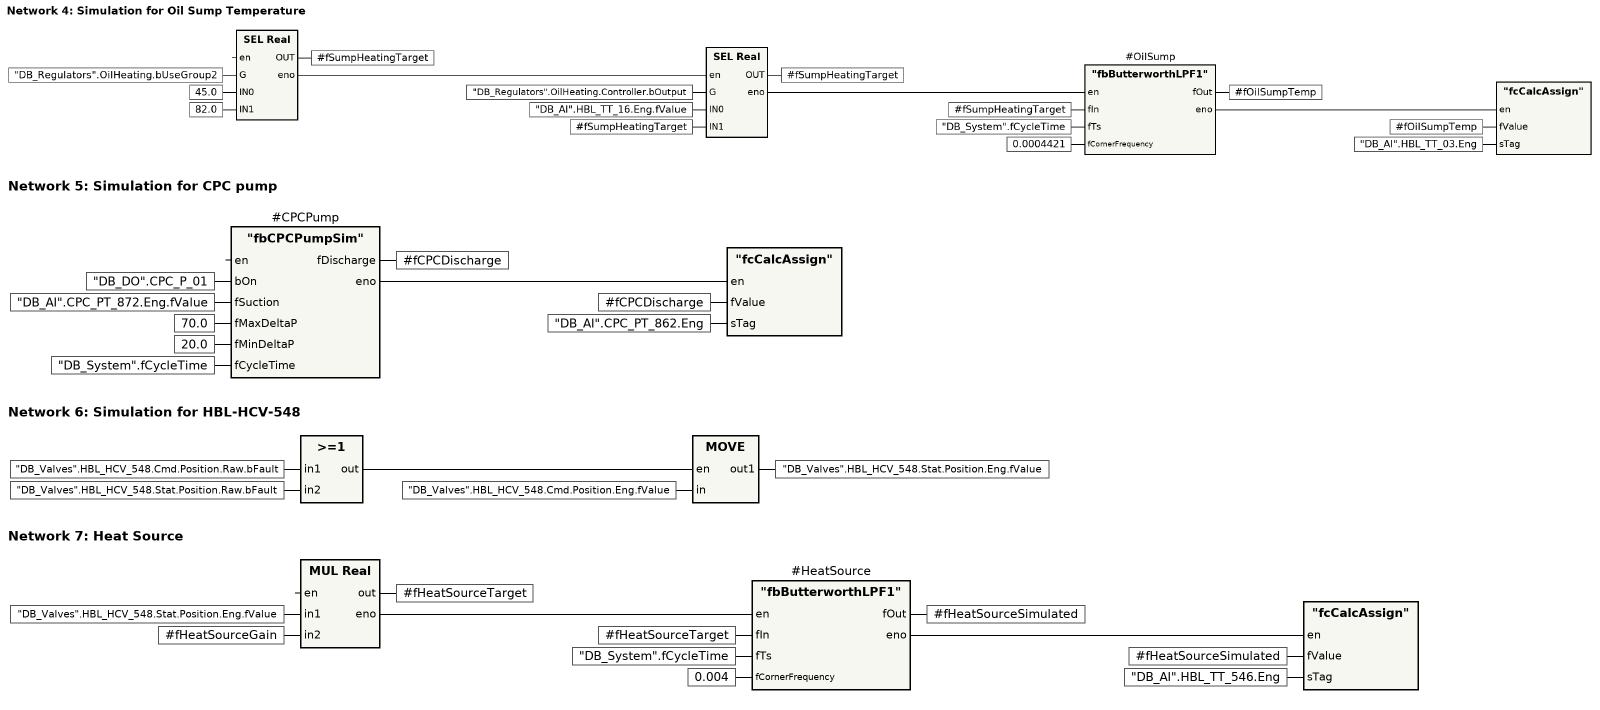
   // ENO of a box is taken as its EN; it also drops when the box reports an error
   #fSumpHeatingTarget := SEL(G := "DB_Regulators".OilHeating.bUseGroup2, IN0 := 45.0, IN1 := 82.0);
   #fSumpHeatingTarget := SEL(G := "DB_Regulators".OilHeating.Controller.bOutput, IN0 := "DB_AI".HBL_TT_16.Eng.fValue, IN1 := #fSumpHeatingTarget);
   #OilSump(fIn := #fSumpHeatingTarget,   // "fbButterworthLPF1"
            fTs := "DB_System".fCycleTime,
            fCornerFrequency := 0.0004421,
            fOut => #fOilSumpTemp,
            ENO => #_w1);
   IF #_w1 THEN "fcCalcAssign"(fValue := #fOilSumpTemp, sTag := "DB_AI".HBL_TT_03.Eng); END_IF;
END_REGION

REGION Network 5: Simulation for CPC pump
   #CPCPump(bOn := "DB_DO".CPC_P_01,   // "fbCPCPumpSim"
            fSuction := "DB_AI".CPC_PT_872.Eng.fValue,
            fMaxDeltaP := 70.0,
            fMinDeltaP := 20.0,
            fCycleTime := "DB_System".fCycleTime,
            fDischarge => #fCPCDischarge,
            ENO => #_w1);
   IF #_w1 THEN "fcCalcAssign"(fValue := #fCPCDischarge, sTag := "DB_AI".CPC_PT_862.Eng); END_IF;
END_REGION

REGION Network 6: Simulation for HBL-HCV-548
   // Only overwrite if the valve is not simulated electrically
   IF "DB_Valves".HBL_HCV_548.Cmd.Position.Raw.bFault OR "DB_Valves".HBL_HCV_548.Stat.Position.Raw.bFault THEN
       "DB_Valves".HBL_HCV_548.Stat.Position.Eng.fValue := "DB_Valves".HBL_HCV_548.Cmd.Position.Eng.fValue;
   END_IF;
END_REGION

REGION Network 7: Heat Source
   // Simulate heat source suction temperature
   #fHeatSourceTarget := "DB_Valves".HBL_HCV_548.Stat.Position.Eng.fValue * #fHeatSourceGain;
   #HeatSource(fIn := #fHeatSourceTarget,   // "fbButterworthLPF1"
               fTs := "DB_System".fCycleTime,
               fCornerFrequency := 0.004,
               fOut => #fHeatSourceSimulated,
               ENO => #_w1);
   IF #_w1 THEN "fcCalcAssign"(fValue := #fHeatSourceSimulated, sTag := "DB_AI".HBL_TT_546.Eng); END_IF;
END_REGION
END_FUNCTION_BLOCK

FUNCTION_BLOCK "fbButterworthLPF1"
{ S7_Optimized_Access := 'TRUE' }
AUTHOR : Heaten
VERSION : 0.1
   VAR_INPUT 
      fIn : Real;   // Value to be filtered (x[n])
      fTs : Real;   // [s]
      fCornerFrequency : Real;   // [Hz]
   END_VAR

   VAR_OUTPUT 
      fOut : Real;   // Filtered value (y[n])
   END_VAR

   VAR 
      fOutPrev : Real;   // y[n-1]
      A : Real;   // [1] Filter coefficient
   END_VAR

   VAR_TEMP 
      tau : Real;   // [s] Filter time constant
      Ts : Real;   // [s] Sampling time
   END_VAR

   VAR CONSTANT 
      PI : Real := 3.141529;
   END_VAR


BEGIN
	// First-order Butterworth IIR filter
	// y[n] = y[n-1] + A*(x[n] - y[n-1])
	// A = Ts / (Ts + RC)
	// Ts = 1/fs
	// RC = 1/(2*pi*fc) = tau
	// 
	// Notes:
	//  - can be used to simulate a first-order process like heating & cooling
	//  - probably some limitation to the corner frequency with respect to the sampling frequency. 10:1 has been mentioned in the literature
	
	// For now, calculate the filter coefficient on every cycle, though it only needs to be done on change or with a bInit input pin
	#tau := 1 / (2 * #PI * #fCornerFrequency);
	#Ts := #fTs;
	#A := #Ts / (#Ts + #tau);
	
	// Filter
	#fOut := #fOutPrev + #A * (#fIn - #fOutPrev);
	
	#fOutPrev := #fOut;
	
END_FUNCTION_BLOCK

FUNCTION_BLOCK "fbCPCPumpSim"   // FB51, FBD
TITLE = CPC pump simulator
{ S7_Optimized_Access := 'TRUE' }
AUTHOR : Heaten
VERSION : 0.1
// stored: AutoNumber true, IsIECCheckEnabled false, IsRetainMemResEnabled false, MemoryReserve 100, SetENOAutomatically false, UDAEnableTagReadback false
   VAR_INPUT
      bOn : Bool;
      fSuction : Real;   // [kPa]
      fMaxDeltaP : Real;   // [kPa]
      fMinDeltaP : Real;   // [kPa]
      fCycleTime : Real;
   END_VAR
   VAR_OUTPUT
      fDischarge : Real;   // [kPa]
   END_VAR
   VAR
      fDeltaP : Real;   // Pressure rise over the pump
      eOn : R_TRIG;
   END_VAR
BEGIN

REGION Network 1: Preset pressure to max at pump start
